(* Logix 5000 project; controller NSH_PLC2 vendor 1 type 14 code 167 rev 32.14; software revision 32.03 *)
// North State Hulling, PLC #2. Passes MCC#2 & #3 Motor Status & control to PLC #1

TASK MainTask (continuous, watchdog 500 ms) : MainProgram

MODULES
   Local : vendor 1 type 14 code 167 (ICP 1, Ethernet 192.168.2.253, rev 32.14)
      NSH_PLC1 : vendor 1 type 14 code 167 (ICP 0, rev 32.1)
      AOP_MCC3_3K : PowerFlex 525-EENET (Ethernet 192.168.3.10, rev 5.2, Output RPI 250 ms)
          : vendor 1 type 150 code 33279 (DSI 1, rev 3.1)
      AOP_MCC3_8K : PowerFlex 525-EENET (Ethernet 192.168.3.33, rev 5.2, Output RPI 250 ms)
          : vendor 1 type 150 code 33279 (DSI 1, rev 3.1)
      AOP_MCC2_21K : PowerFlex 525-EENET (Ethernet 192.168.2.116, rev 5.2, Output RPI 100 ms)
          : vendor 1 type 150 code 33279 (DSI 1, rev 3.1)
      AOP_MCC3_5K : PowerFlex 525-EENET (Ethernet 192.168.3.18, rev 5.2, Output RPI 250 ms)
          : vendor 1 type 150 code 33279 (DSI 1, rev 3.1)
      AOP_MCC3_2A : PowerFlex 525-EENET (Ethernet 192.168.3.3, rev 5.2, Output RPI 250 ms)
          : vendor 1 type 150 code 33279 (DSI 1, rev 3.1)
      AOP_MCC3_2K : PowerFlex 525-EENET (Ethernet 192.168.3.6, rev 5.2, Output RPI 250 ms)
          : vendor 1 type 150 code 33279 (DSI 1, rev 3.1)
      AOP_MCC3_3G : PowerFlex 525-EENET (Ethernet 192.168.3.9, rev 5.2, Output RPI 250 ms)
          : vendor 1 type 150 code 33279 (DSI 1, rev 3.1)
      AOP_MCC4_1E : PowerFlex 525-EENET (Ethernet 192.168.3.150, rev 6.1, Output RPI 100 ms)
          : vendor 1 type 150 code 33279 (DSI 1, rev 3.1)
      AOP_MCC3_4A : PowerFlex 525-EENET (Ethernet 192.168.3.11, rev 5.2, Output RPI 250 ms)
          : vendor 1 type 150 code 33279 (DSI 1, rev 3.1)
      AOP_MCC3_2D : PowerFlex 525-EENET (Ethernet 192.168.3.4, rev 5.2, Output RPI 250 ms)
          : vendor 1 type 150 code 33279 (DSI 1, rev 3.1)
      AOP_MCC2_9H : PowerFlex 525-EENET (Ethernet 192.168.2.43, rev 5.2, Output RPI 100 ms)
          : vendor 1 type 150 code 33279 (DSI 1, rev 3.1)
      AOP_MCC2_2K : PowerFlex 525-EENET (Ethernet 192.168.2.6, rev 5.2, Output RPI 250 ms)
          : vendor 1 type 150 code 33279 (DSI 1, rev 3.1)
      AOP_MCC3_4D : PowerFlex 525-EENET (Ethernet 192.168.3.12, rev 5.2, Output RPI 250 ms)
          : vendor 1 type 150 code 33279 (DSI 1, rev 3.1)
      AOP_MCC3_7G : PowerFlex 525-EENET (Ethernet 192.168.3.28, rev 5.2, Output RPI 250 ms)
          : vendor 1 type 150 code 33279 (DSI 1, rev 3.1)
      AOP_MCC3_3D : PowerFlex 525-EENET (Ethernet 192.168.3.8, rev 5.2, Output RPI 250 ms)
          : vendor 1 type 150 code 33279 (DSI 1, rev 3.1)
      AOP_MCC3_6D : PowerFlex 525-EENET (Ethernet 192.168.3.20, rev 5.2, Output RPI 250 ms)
          : vendor 1 type 150 code 33279 (DSI 1, rev 3.1)
      AOP_MCC4_2K : PowerFlex 525-EENET (Ethernet 192.168.3.155, rev 6.1, Output RPI 100 ms)
          : vendor 1 type 150 code 33279 (DSI 1, rev 3.1)
      AOP_MCC3_5G : PowerFlex 525-EENET (Ethernet 192.168.3.17, rev 5.2, Output RPI 250 ms)
          : vendor 1 type 150 code 33279 (DSI 1, rev 3.1)
      AOP_MCC3_6A : PowerFlex 525-EENET (Ethernet 192.168.3.19, rev 5.2, Output RPI 250 ms)
          : vendor 1 type 150 code 33279 (DSI 1, rev 3.1)
      AOP_MCC3_5D : PowerFlex 525-EENET (Ethernet 192.168.3.16, rev 5.2, Output RPI 250 ms)
      AOP_MCC2_2G : PowerFlex 525-EENET (Ethernet 192.168.2.5, rev 5.2, Output RPI 250 ms)
          : vendor 1 type 150 code 33279 (DSI 1, rev 3.1)
      AOP_MCC3_5A : PowerFlex 525-EENET (Ethernet 192.168.3.15, rev 5.2, Output RPI 250 ms)
          : vendor 1 type 150 code 33279 (DSI 1, rev 3.1)
      AOP_MCC3_7K : PowerFlex 525-EENET (Ethernet 192.168.3.29, rev 5.2, Output RPI 250 ms)
          : vendor 1 type 150 code 33279 (DSI 1, rev 3.1)
      AOP_MCC2_21G : PowerFlex 525-EENET (Ethernet 192.168.2.115, rev 5.2, Output RPI 250 ms)
          : vendor 1 type 150 code 33279 (DSI 1, rev 3.1)
      AOP_MCC3_2G : PowerFlex 525-EENET (Ethernet 192.168.3.5, rev 5.2, Output RPI 250 ms)
          : vendor 1 type 150 code 33279 (DSI 1, rev 3.1)
      AOP_MCC3_4G : PowerFlex 525-EENET (Ethernet 192.168.3.13, rev 5.2, Output RPI 250 ms)
          : vendor 1 type 150 code 33279 (DSI 1, rev 3.1)
      AOP_MCC2_2A : PowerFlex 525-EENET (Ethernet 192.168.2.3, rev 5.2, Output RPI 250 ms)
          : vendor 1 type 150 code 33279 (DSI 1, rev 3.1)
      AOP_MCC2_2D : PowerFlex 525-EENET (Ethernet 192.168.2.4, rev 5.2, Output RPI 250 ms)
          : vendor 1 type 150 code 33279 (DSI 1, rev 3.1)
      AOP_MCC3_8D : PowerFlex 525-EENET (Ethernet 192.168.3.31, rev 5.2, Output RPI 250 ms)
          : vendor 1 type 150 code 33279 (DSI 1, rev 3.1)
      AOP_MCC3_3A : PowerFlex 525-EENET (Ethernet 192.168.3.7, rev 5.2, Output RPI 250 ms)
          : vendor 1 type 150 code 33279 (DSI 1, rev 3.1)
      AOP_MCC4_2G : PowerFlex 525-EENET (Ethernet 192.168.3.154, rev 5.2, Output RPI 100 ms)
          : vendor 1 type 150 code 33279 (DSI 1, rev 3.1)
      AOP_MCC3_4K : PowerFlex 525-EENET (Ethernet 192.168.3.14, rev 5.2, Output RPI 250 ms)
          : vendor 1 type 150 code 33279 (DSI 1, rev 3.1)
      AOP_MCC2_13L_1 : vendor 1 type 12 code 237 (Ethernet 192.168.2.204, rev 10.1, Output RPI 1000 ms)
      AOP_MCC4_1L_1 : vendor 1 type 12 code 237 (Ethernet 192.168.3.210, rev 10.1, Output RPI 1000 ms)
      AOP_MCC2_9L_2 : vendor 1 type 12 code 243 (Ethernet 192.168.2.203, rev 10.1, Output RPI 1000 ms)
      AOP_MCC3_10L_2 : vendor 1 type 12 code 243 (Ethernet 192.168.3.203, rev 10.1, Output RPI 1000 ms)
      AOP_MCC3_15L_1 : vendor 1 type 12 code 237 (Ethernet 192.168.3.204, rev 10.1, Output RPI 1000 ms)
      AOP_MCC2_13L_2 : vendor 1 type 12 code 243 (Ethernet 192.168.2.205, rev 10.1, Output RPI 1000 ms)
      AOP_MCC3_15L_2 : vendor 1 type 12 code 243 (Ethernet 192.168.3.205, rev 10.1, Output RPI 1000 ms)
      AOP_MCC4_1L_2 : vendor 1 type 12 code 243 (Ethernet 192.168.3.211, rev 10.1, Output RPI 1000 ms)
      AOP_MCC2_5L_1 : vendor 1 type 12 code 237 (Ethernet 192.168.2.200, rev 10.1, Output RPI 1000 ms)
      AOP_MCC3_6L_2 : vendor 1 type 12 code 243 (Ethernet 192.168.3.201, rev 10.1, Output RPI 1000 ms)
      AOP_MCC3_20L_1 : vendor 1 type 12 code 237 (Ethernet 192.168.3.208, rev 10.1, Output RPI 1000 ms)
      AOP_MCC2_9L_1 : vendor 1 type 12 code 237 (Ethernet 192.168.2.202, rev 10.1, Output RPI 1000 ms)
      AOP_MCC2_20L_2 : vendor 1 type 12 code 243 (Ethernet 192.168.2.209, rev 10.1, Output RPI 1000 ms)
      AOP_MCC3_19L_2 : vendor 1 type 12 code 243 (Ethernet 192.168.3.207, rev 10.1, Output RPI 1000 ms)
      AOP_MCC3_20L_2 : vendor 1 type 12 code 243 (Ethernet 192.168.3.209, rev 10.1, Output RPI 1000 ms)
      AOP_MCC2_5L_2 : vendor 1 type 12 code 243 (Ethernet 192.168.2.201, rev 10.1, Output RPI 1000 ms)
      AOP_MCC2_20L_1 : vendor 1 type 12 code 237 (Ethernet 192.168.2.208, rev 10.1, Output RPI 1000 ms)
      AOP_MCC3_6L_1 : vendor 1 type 12 code 237 (Ethernet 192.168.3.200, rev 10.1, Output RPI 1000 ms)
      AOP_MCC2_17L_2 : vendor 1 type 12 code 243 (Ethernet 192.168.2.207, rev 10.1, Output RPI 1000 ms)
      AOP_MCC2_17L_1 : vendor 1 type 12 code 237 (Ethernet 192.168.2.206, rev 10.1, Output RPI 1000 ms)
      AOP_MCC3_19L_1 : vendor 1 type 12 code 237 (Ethernet 192.168.3.206, rev 10.1, Output RPI 1000 ms)
      AOP_MCC3_10L_1 : vendor 1 type 12 code 237 (Ethernet 192.168.3.202, rev 10.1, Output RPI 1000 ms)
      AOP_MCC3_16G : 193-ECM-ETR (Ethernet 192.168.3.78, rev 7.17, StandardDataDriven RPI 100 ms)
      AOP_MCC2_4C : 193-ECM-ETR (Ethernet 192.168.2.14, rev 7.17, StandardDataDriven RPI 100 ms)
      AOP_MCC2_21E : 193-ECM-ETR (Ethernet 192.168.2.114, rev 7.17, StandardDataDriven RPI 100 ms)
      AOP_MCC3_13C : 193-ECM-ETR (Ethernet 192.168.3.57, rev 7.17, StandardDataDriven RPI 100 ms)
      AOP_MCC3_18C : 193-ECM-ETR (Ethernet 192.168.3.88, rev 7.17, StandardDataDriven RPI 100 ms)
      AOP_MCC3_13A : 193-ECM-ETR (Ethernet 192.168.3.56, rev 7.17, StandardDataDriven RPI 100 ms)
      AOP_MCC3_15C : 193-ECM-ETR (Ethernet 192.168.3.69, rev 7.17, StandardDataDriven RPI 100 ms)
      AOP_MCC3_6G : 193-ECM-ETR (Ethernet 192.168.3.21, rev 7.17, StandardDataDriven RPI 100 ms)
      AOP_MCC2_4L : 193-ECM-ETR (Ethernet 192.168.2.18, rev 7.17, StandardDataDriven RPI 100 ms)
      AOP_MCC3_11A : 193-ECM-ETR (Ethernet 192.168.3.44, rev 7.17, StandardDataDriven RPI 100 ms)
      AOP_MCC2_10A : 193-ECM-ETR (Ethernet 192.168.2.46, rev 7.17, StandardDataDriven RPI 100 ms)
      AOP_MCC2_13J : 193-ECM-ETR (Ethernet 192.168.2.68, rev 7.17, StandardDataDriven RPI 100 ms)
      AOP_MCC4_4A : 193-ECM-ETR (Ethernet 192.168.3.162, rev 7.17, StandardDataDriven RPI 100 ms)
      AOP_MCC2_4G : 193-ECM-ETR (Ethernet 192.168.2.16, rev 7.17, StandardDataDriven RPI 100 ms)
      AOP_MCC2_8D : 193-ECM-ETR (Ethernet 192.168.2.37, rev 7.17, StandardDataDriven RPI 100 ms)
      AOP_MCC4_5C : 193-ECM-ETR (Ethernet 192.168.3.169, rev 7.17, StandardDataDriven RPI 100 ms)
      AOP_MCC3_16E : 193-ECM-ETR (Ethernet 192.168.3.77, rev 7.17, StandardDataDriven RPI 100 ms)
      AOP_MCC3_10J : 193-ECM-ETR (Ethernet 192.168.3.43, rev 7.17, StandardDataDriven RPI 100 ms)
      AOP_MCC2_3A : 193-ECM-ETR (Ethernet 192.168.2.7, rev 7.17, StandardDataDriven RPI 100 ms)
      AOP_MCC3_13G : 193-ECM-ETR (Ethernet 192.168.3.59, rev 7.17, StandardDataDriven RPI 100 ms)
      AOP_MCC2_3C : 193-ECM-ETR (Ethernet 192.168.2.8, rev 7.17, StandardDataDriven RPI 100 ms)
      AOP_MCC3_12G : 193-ECM-ETR (Ethernet 192.168.3.53, rev 7.17, StandardDataDriven RPI 100 ms)
      AOP_MCC4_4L : 193-ECM-ETR (Ethernet 192.168.3.167, rev 7.17, StandardDataDriven RPI 100 ms)
      AOP_MCC2_14E : 193-ECM-ETR (Ethernet 192.168.2.73, rev 7.17, StandardDataDriven RPI 100 ms)
      AOP_MCC3_21C : 193-ECM-ETR (Ethernet 192.168.3.106, rev 7.17, StandardDataDriven RPI 100 ms)
      AOP_MCC3_21E : 193-ECM-ETR (Ethernet 192.168.3.107, rev 7.17, StandardDataDriven RPI 100 ms)
      AOP_MCC3_20G : 193-ECM-ETR (Ethernet 192.168.3.103, rev 7.17, StandardDataDriven RPI 100 ms)
      AOP_MCC2_12J : 193-ECM-ETR (Ethernet 192.168.2.62, rev 7.17, StandardDataDriven RPI 100 ms)
      AOP_MCC3_12J : 193-ECM-ETR (Ethernet 192.168.3.54, rev 7.17, StandardDataDriven RPI 100 ms)
      AOP_MCC3_15E : 193-ECM-ETR (Ethernet 192.168.3.70, rev 7.17, StandardDataDriven RPI 100 ms)
      AOP_MCC3_19C : 193-ECM-ETR (Ethernet 192.168.3.94, rev 7.17, StandardDataDriven RPI 100 ms)
      AOP_MCC4_4G : 193-ECM-ETR (Ethernet 192.168.3.165, rev 7.17, StandardDataDriven RPI 100 ms)
      AOP_MCC3_8H : 193-ECM-ETR (Ethernet 192.168.3.32, rev 7.17, StandardDataDriven RPI 100 ms)
      AOP_MCC2_11G : 193-ECM-ETR (Ethernet 192.168.2.55, rev 7.17, StandardDataDriven RPI 100 ms)
      AOP_MCC2_17C : 193-ECM-ETR (Ethernet 192.168.2.90, rev 7.17, StandardDataDriven RPI 100 ms)
      AOP_MCC3_14G : 193-ECM-ETR (Ethernet 192.168.3.65, rev 7.17, StandardDataDriven RPI 100 ms)
      AOP_MCC4_2A : 193-ECM-ETR (Ethernet 192.168.3.151, rev 7.17, StandardDataDriven RPI 100 ms)
      AOP_MCC3_22E : 193-ECM-ETR (Ethernet 192.168.3.112, rev 7.17, StandardDataDriven RPI 100 ms)
      AOP_MCC3_15G : 193-ECM-ETR (Ethernet 192.168.3.71, rev 7.17, StandardDataDriven RPI 100 ms)
      AOP_MCC2_13C : 193-ECM-ETR (Ethernet 192.168.2.65, rev 7.17, StandardDataDriven RPI 100 ms)
      AOP_MCC2_3J : 193-ECM-ETR (Ethernet 192.168.2.11, rev 7.17, StandardDataDriven RPI 100 ms)
      AOP_MCC3_17G : 193-ECM-ETR (Ethernet 192.168.3.84, rev 7.17, StandardDataDriven RPI 250 ms)
      AOP_MCC3_17A : 193-ECM-ETR (Ethernet 192.168.3.81, rev 7.17, StandardDataDriven RPI 100 ms)
      AOP_MCC3_19A : 193-ECM-ETR (Ethernet 192.168.3.93, rev 7.17, StandardDataDriven RPI 100 ms)
      AOP_MCC2_16E : 193-ECM-ETR (Ethernet 192.168.2.85, rev 7.17, StandardDataDriven RPI 100 ms)
      AOP_MCC2_10C : 193-ECM-ETR (Ethernet 192.168.2.47, rev 7.17, StandardDataDriven RPI 100 ms)
      AOP_MCC3_21G : 193-ECM-ETR (Ethernet 192.168.3.108, rev 7.17, StandardDataDriven RPI 100 ms)
      AOP_MCC2_8H : 193-ECM-ETR (Ethernet 192.168.2.39, rev 7.17, StandardDataDriven RPI 100 ms)
      AOP_MCC2_6C : 193-ECM-ETR (Ethernet 192.168.2.27, rev 7.17, StandardDataDriven RPI 100 ms)
      AOP_MCC4_3G : 193-ECM-ETR (Ethernet 192.168.3.159, rev 7.17, StandardDataDriven RPI 100 ms)
      AOP_MCC2_16C : 193-ECM-ETR (Ethernet 192.168.2.84, rev 7.17, StandardDataDriven RPI 100 ms)
      AOP_MCC3_18G : 193-ECM-ETR (Ethernet 192.168.3.90, rev 7.17, StandardDataDriven RPI 100 ms)
      AOP_MCC2_8F : 193-ECM-ETR (Ethernet 192.168.2.38, rev 7.17, StandardDataDriven RPI 100 ms)
      AOP_MCC2_13E : 193-ECM-ETR (Ethernet 192.168.2.66, rev 7.17, StandardDataDriven RPI 100 ms)
      AOP_MCC3_12L : 193-ECM-ETR (Ethernet 192.168.3.55, rev 7.17, StandardDataDriven RPI 100 ms)
      AOP_MCC2_18J : 193-ECM-ETR (Ethernet 192.168.2.100, rev 7.17, StandardDataDriven RPI 100 ms)
      AOP_MCC2_20J : 193-ECM-ETR (Ethernet 192.168.2.111, rev 7.17, StandardDataDriven RPI 100 ms)
      AOP_MCC2_15G : 193-ECM-ETR (Ethernet 192.168.2.80, rev 7.17, StandardDataDriven RPI 100 ms)
      AOP_MCC3_19G : 193-ECM-ETR (Ethernet 192.168.3.96, rev 7.17, StandardDataDriven RPI 100 ms)
      AOP_MCC4_2E : 193-ECM-ETR (Ethernet 192.168.3.153, rev 7.17, StandardDataDriven RPI 100 ms)
      AOP_MCC2_19C : 193-ECM-ETR (Ethernet 192.168.2.103, rev 7.17, StandardDataDriven RPI 100 ms)
      AOP_MCC2_15J : 193-ECM-ETR (Ethernet 192.168.2.81, rev 7.17, StandardDataDriven RPI 100 ms)
      AOP_MCC3_12A : 193-ECM-ETR (Ethernet 192.168.3.50, rev 7.17, StandardDataDriven RPI 100 ms)
      AOP_MCC3_11G : 193-ECM-ETR (Ethernet 192.168.3.46, rev 7.17, StandardDataDriven RPI 100 ms)
      AOP_MCC3_13L : 193-ECM-ETR (Ethernet 192.168.3.61, rev 7.17, StandardDataDriven RPI 100 ms)
      AOP_MCC2_11J : 193-ECM-ETR (Ethernet 192.168.2.56, rev 7.17, StandardDataDriven RPI 100 ms)
      AOP_MCC3_6J : 193-ECM-ETR (Ethernet 192.168.3.22, rev 7.17, StandardDataDriven RPI 100 ms)
      AOP_MCC3_10G : 193-ECM-ETR (Ethernet 192.168.3.42, rev 7.17, StandardDataDriven RPI 100 ms)
      AOP_MCC2_16L : 193-ECM-ETR (Ethernet 192.168.2.88, rev 7.17, StandardDataDriven RPI 100 ms)
      AOP_MCC2_18C : 193-ECM-ETR (Ethernet 192.168.2.97, rev 7.17, StandardDataDriven RPI 100 ms)
      AOP_MCC2_14G : 193-ECM-ETR (Ethernet 192.168.2.74, rev 7.17, StandardDataDriven RPI 100 ms)
      AOP_MCC2_7G : 193-ECM-ETR (Ethernet 192.168.2.34, rev 7.17, StandardDataDriven RPI 100 ms)
      AOP_MCC2_19E : 193-ECM-ETR (Ethernet 192.168.2.104, rev 7.17, StandardDataDriven RPI 100 ms)
      AOP_MCC2_15E : 193-ECM-ETR (Ethernet 192.168.2.79, rev 7.17, StandardDataDriven RPI 100 ms)
      AOP_MCC3_21A : 193-ECM-ETR (Ethernet 192.168.3.105, rev 7.17, StandardDataDriven RPI 100 ms)
      AOP_MCC2_5G : 193-ECM-ETR (Ethernet 192.168.2.22, rev 7.17, StandardDataDriven RPI 100 ms)
      AOP_MCC3_18L : 193-ECM-ETR (Ethernet 192.168.3.92, rev 7.17, StandardDataDriven RPI 100 ms)
      AOP_MCC2_10E : 193-ECM-ETR (Ethernet 192.168.2.48, rev 7.17, StandardDataDriven RPI 100 ms)
      AOP_MCC2_3G : 193-ECM-ETR (Ethernet 192.168.2.10, rev 7.17, StandardDataDriven RPI 100 ms)
      AOP_MCC3_16J : 193-ECM-ETR (Ethernet 192.168.3.79, rev 7.17, StandardDataDriven RPI 100 ms)
      AOP_MCC3_7E : 193-ECM-ETR (Ethernet 192.168.3.27, rev 7.17, StandardDataDriven RPI 100 ms)
      AOP_MCC2_13A : 193-ECM-ETR (Ethernet 192.168.2.64, rev 7.17, StandardDataDriven RPI 100 ms)
      AOP_MCC3_19J : 193-ECM-ETR (Ethernet 192.168.3.97, rev 7.17, StandardDataDriven RPI 100 ms)
      AOP_MCC3_21J : 193-ECM-ETR (Ethernet 192.168.3.109, rev 7.17, StandardDataDriven RPI 100 ms)
      AOP_MCC2_13G : 193-ECM-ETR (Ethernet 192.168.2.67, rev 7.17, StandardDataDriven RPI 100 ms)
      AOP_MCC2_7K : 193-ECM-ETR (Ethernet 192.168.2.35, rev 7.17, StandardDataDriven RPI 100 ms)
      AOP_MCC3_20C : 193-ECM-ETR (Ethernet 192.168.3.101, rev 7.17, StandardDataDriven RPI 100 ms)
      AOP_MCC2_18L : 193-ECM-ETR (Ethernet 192.168.2.101, rev 7.17, StandardDataDriven RPI 100 ms)
      AOP_MCC2_3E : 193-ECM-ETR (Ethernet 192.168.2.9, rev 7.17, StandardDataDriven RPI 100 ms)
      AOP_MCC2_6L : 193-ECM-ETR (Ethernet 192.168.2.31, rev 7.17, StandardDataDriven RPI 100 ms)
      AOP_MCC2_16A : 193-ECM-ETR (Ethernet 192.168.2.83, rev 7.17, StandardDataDriven RPI 100 ms)
      AOP_MCC3_9L : 193-ECM-ETR (Ethernet 192.168.3.39, rev 7.17, StandardDataDriven RPI 100 ms)
      AOP_MCC2_12A : 193-ECM-ETR (Ethernet 192.168.2.58, rev 7.17, StandardDataDriven RPI 100 ms)
      AOP_MCC3_18J : 193-ECM-ETR (Ethernet 192.168.3.91, rev 7.17, StandardDataDriven RPI 100 ms)
      AOP_MCC4_4J : 193-ECM-ETR (Ethernet 192.168.3.166, rev 7.17, StandardDataDriven RPI 100 ms)
      AOP_MCC3_14L : 193-ECM-ETR (Ethernet 192.168.3.67, rev 7.17, StandardDataDriven RPI 100 ms)
      AOP_MCC3_12C : 193-ECM-ETR (Ethernet 192.168.3.51, rev 7.17, StandardDataDriven RPI 100 ms)
      AOP_MCC2_3L : 193-ECM-ETR (Ethernet 192.168.2.12, rev 7.17, StandardDataDriven RPI 100 ms)
      AOP_MCC3_9G : 193-ECM-ETR (Ethernet 192.168.3.37, rev 7.17, StandardDataDriven RPI 100 ms)
      AOP_MCC3_17C : 193-ECM-ETR (Ethernet 192.168.3.82, rev 7.17, StandardDataDriven RPI 100 ms)
      AOP_MCC3_17L : 193-ECM-ETR (Ethernet 192.168.3.86, rev 7.17, StandardDataDriven RPI 100 ms)
      AOP_MCC4_4C : 193-ECM-ETR (Ethernet 192.168.3.163, rev 7.17, StandardDataDriven RPI 100 ms)
      AOP_MCC2_4E : 193-ECM-ETR (Ethernet 192.168.2.15, rev 7.17, StandardDataDriven RPI 100 ms)
      AOP_MCC3_9C : 193-ECM-ETR (Ethernet 192.168.3.35, rev 7.17, StandardDataDriven RPI 100 ms)
      AOP_MCC2_17A : 193-ECM-ETR (Ethernet 192.168.2.89, rev 7.17, StandardDataDriven RPI 100 ms)
      AOP_MCC3_9E : 193-ECM-ETR (Ethernet 192.168.3.36, rev 7.17, StandardDataDriven RPI 100 ms)
      AOP_MCC3_18E : 193-ECM-ETR (Ethernet 192.168.3.89, rev 7.17, StandardDataDriven RPI 100 ms)
      AOP_MCC2_11C : 193-ECM-ETR (Ethernet 192.168.2.53, rev 7.17, StandardDataDriven RPI 100 ms)
      AOP_MCC2_18E : 193-ECM-ETR (Ethernet 192.168.2.98, rev 7.17, StandardDataDriven RPI 100 ms)
      AOP_MCC2_5A : 193-ECM-ETR (Ethernet 192.168.2.19, rev 7.17, StandardDataDriven RPI 100 ms)
      AOP_MCC3_16L : 193-ECM-ETR (Ethernet 192.168.3.80, rev 7.17, StandardDataDriven RPI 100 ms)
      AOP_MCC2_19J : 193-ECM-ETR (Ethernet 192.168.2.106, rev 7.17, StandardDataDriven RPI 100 ms)
      AOP_MCC2_10G : 193-ECM-ETR (Ethernet 192.168.2.49, rev 7.17, StandardDataDriven RPI 100 ms)
      AOP_MCC4_3C : 193-ECM-ETR (Ethernet 192.168.3.157, rev 7.17, StandardDataDriven RPI 100 ms)
      AOP_MCC4_2C : 193-ECM-ETR (Ethernet 192.168.3.152, rev 7.17, StandardDataDriven RPI 100 ms)
      AOP_MCC2_19A : 193-ECM-ETR (Ethernet 192.168.2.102, rev 7.17, StandardDataDriven RPI 100 ms)
      AOP_MCC2_20G : 193-ECM-ETR (Ethernet 192.168.2.110, rev 7.17, StandardDataDriven RPI 100 ms)
      AOP_MCC3_14J : 193-ECM-ETR (Ethernet 192.168.3.66, rev 7.17, StandardDataDriven RPI 100 ms)
      AOP_MCC2_10L : 193-ECM-ETR (Ethernet 192.168.2.51, rev 7.17, StandardDataDriven RPI 100 ms)
      AOP_MCC3_15A : 193-ECM-ETR (Ethernet 192.168.3.68, rev 7.17, StandardDataDriven RPI 100 ms)
      AOP_MCC2_14L : 193-ECM-ETR (Ethernet 192.168.2.76, rev 7.17, StandardDataDriven RPI 100 ms)
      AOP_MCC4_3E : 193-ECM-ETR (Ethernet 192.168.3.158, rev 7.17, StandardDataDriven RPI 100 ms)
      AOP_MCC2_19L : 193-ECM-ETR (Ethernet 192.168.2.107, rev 7.17, StandardDataDriven RPI 100 ms)
      AOP_MCC2_17J : 193-ECM-ETR (Ethernet 192.168.2.93, rev 7.17, StandardDataDriven RPI 100 ms)
      AOP_MCC3_14A : 193-ECM-ETR (Ethernet 192.168.3.62, rev 7.17, StandardDataDriven RPI 100 ms)
      AOP_MCC3_14E : 193-ECM-ETR (Ethernet 192.168.3.64, rev 7.17, StandardDataDriven RPI 100 ms)
      AOP_MCC2_4A : 193-ECM-ETR (Ethernet 192.168.2.13, rev 7.17, StandardDataDriven RPI 100 ms)
      AOP_MCC4_4E : 193-ECM-ETR (Ethernet 192.168.3.164, rev 7.17, StandardDataDriven RPI 100 ms)
      AOP_MCC2_10J : 193-ECM-ETR (Ethernet 192.168.2.50, rev 7.17, StandardDataDriven RPI 100 ms)
      AOP_MCC3_20A : 193-ECM-ETR (Ethernet 192.168.3.100, rev 7.17, StandardDataDriven RPI 100 ms)
      AOP_MCC2_6G : 193-ECM-ETR (Ethernet 192.168.2.29, rev 7.17, StandardDataDriven RPI 100 ms)
      AOP_MCC3_16A : 193-ECM-ETR (Ethernet 192.168.3.75, rev 7.17, StandardDataDriven RPI 100 ms)
      AOP_MCC2_14J : 193-ECM-ETR (Ethernet 192.168.2.75, rev 7.17, StandardDataDriven RPI 100 ms)
      AOP_MCC2_6A : 193-ECM-ETR (Ethernet 192.168.2.26, rev 7.17, StandardDataDriven RPI 100 ms)
      AOP_MCC2_17G : 193-ECM-ETR (Ethernet 192.168.2.92, rev 7.17, StandardDataDriven RPI 100 ms)
      AOP_MCC2_17E : 193-ECM-ETR (Ethernet 192.168.2.91, rev 7.17, StandardDataDriven RPI 100 ms)
      AOP_MCC2_20C : 193-ECM-ETR (Ethernet 192.168.2.108, rev 7.17, StandardDataDriven RPI 100 ms)
      AOP_MCC3_18A : 193-ECM-ETR (Ethernet 192.168.3.87, rev 7.17, StandardDataDriven RPI 100 ms)
      AOP_MCC2_6J : 193-ECM-ETR (Ethernet 192.168.2.30, rev 7.17, StandardDataDriven RPI 100 ms)
      AOP_MCC3_17J : 193-ECM-ETR (Ethernet 192.168.3.85, rev 7.17, StandardDataDriven RPI 100 ms)
      AOP_MCC2_12L : 193-ECM-ETR (Ethernet 192.168.2.63, rev 7.17, StandardDataDriven RPI 100 ms)
      AOP_MCC2_15L : 193-ECM-ETR (Ethernet 192.168.2.82, rev 7.17, StandardDataDriven RPI 100 ms)
      AOP_MCC3_19E : 193-ECM-ETR (Ethernet 192.168.3.95, rev 7.17, StandardDataDriven RPI 100 ms)
      AOP_MCC2_8K : 193-ECM-ETR (Ethernet 192.168.2.40, rev 7.17, StandardDataDriven RPI 250 ms)
      AOP_MCC3_21L : 193-ECM-ETR (Ethernet 192.168.3.110, rev 7.17, StandardDataDriven RPI 100 ms)
      AOP_MCC2_11A : 193-ECM-ETR (Ethernet 192.168.2.52, rev 7.17, StandardDataDriven RPI 100 ms)
      AOP_MCC2_14C : 193-ECM-ETR (Ethernet 192.168.2.72, rev 7.17, StandardDataDriven RPI 100 ms)
      AOP_MCC2_14A : 193-ECM-ETR (Ethernet 192.168.2.71, rev 7.17, StandardDataDriven RPI 100 ms)
      AOP_MCC2_4J : 193-ECM-ETR (Ethernet 192.168.2.17, rev 7.17, StandardDataDriven RPI 100 ms)
      AOP_MCC2_11E : 193-ECM-ETR (Ethernet 192.168.2.54, rev 7.17, StandardDataDriven RPI 100 ms)
      AOP_MCC2_6E : 193-ECM-ETR (Ethernet 192.168.2.28, rev 7.17, StandardDataDriven RPI 100 ms)
      AOP_MCC2_21C : 193-ECM-ETR (Ethernet 192.168.2.113, rev 7.17, StandardDataDriven RPI 100 ms)
      AOP_MCC3_13J : 193-ECM-ETR (Ethernet 192.168.3.60, rev 7.17, StandardDataDriven RPI 100 ms)
      AOP_MCC3_7C : 193-ECM-ETR (Ethernet 192.168.3.26, rev 7.17, StandardDataDriven RPI 100 ms)
      AOP_MCC3_10A : 193-ECM-ETR (Ethernet 192.168.3.40, rev 7.17, StandardDataDriven RPI 100 ms)
      AOP_MCC2_9F : 193-ECM-ETR (Ethernet 192.168.2.42, rev 7.17, StandardDataDriven RPI 100 ms)
      AOP_MCC2_8B : 193-ECM-ETR (Ethernet 192.168.2.36, rev 7.17, StandardDataDriven RPI 100 ms)
      AOP_MCC3_20E : 193-ECM-ETR (Ethernet 192.168.3.102, rev 7.17, StandardDataDriven RPI 100 ms)
      AOP_MCC3_13E : 193-ECM-ETR (Ethernet 192.168.3.58, rev 7.17, StandardDataDriven RPI 100 ms)
      AOP_MCC3_16C : 193-ECM-ETR (Ethernet 192.168.3.76, rev 7.17, StandardDataDriven RPI 100 ms)
      AOP_MCC2_5E : 193-ECM-ETR (Ethernet 192.168.2.21, rev 7.17, StandardDataDriven RPI 100 ms)
      AOP_MCC3_9A : 193-ECM-ETR (Ethernet 192.168.3.34, rev 7.17, StandardDataDriven RPI 100 ms)
      AOP_MCC2_15A : 193-ECM-ETR (Ethernet 192.168.2.77, rev 7.17, StandardDataDriven RPI 100 ms)
      AOP_MCC2_5C : 193-ECM-ETR (Ethernet 192.168.2.20, rev 7.17, StandardDataDriven RPI 100 ms)
      AOP_MCC2_12G : 193-ECM-ETR (Ethernet 192.168.2.61, rev 7.17, StandardDataDriven RPI 100 ms)
      AOP_MCC3_22C : 193-ECM-ETR (Ethernet 192.168.3.111, rev 7.17, StandardDataDriven RPI 100 ms)
      AOP_MCC2_11L : 193-ECM-ETR (Ethernet 192.168.2.57, rev 7.17, StandardDataDriven RPI 100 ms)
      AOP_MCC2_16J : 193-ECM-ETR (Ethernet 192.168.2.87, rev 7.17, StandardDataDriven RPI 100 ms)
      AOP_MCC2_12C : 193-ECM-ETR (Ethernet 192.168.2.59, rev 7.17, StandardDataDriven RPI 100 ms)
      AOP_MCC4_3A : 193-ECM-ETR (Ethernet 192.168.3.156, rev 7.17, StandardDataDriven RPI 100 ms)
      AOP_MCC2_7D : 193-ECM-ETR (Ethernet 192.168.2.33, rev 7.17, StandardDataDriven RPI 100 ms)
      AOP_MCC3_8A : 193-ECM-ETR (Ethernet 192.168.3.30, rev 7.17, StandardDataDriven RPI 100 ms)
      AOP_MCC2_7A : 193-ECM-ETR (Ethernet 192.168.2.32, rev 7.17, StandardDataDriven RPI 100 ms)
      AOP_MCC2_15C : 193-ECM-ETR (Ethernet 192.168.2.78, rev 7.17, StandardDataDriven RPI 150 ms)
      AOP_MCC2_12E : 193-ECM-ETR (Ethernet 192.168.2.60, rev 7.17, StandardDataDriven RPI 100 ms)
      AOP_MCC2_20E : 193-ECM-ETR (Ethernet 192.168.2.109, rev 7.17, StandardDataDriven RPI 100 ms)
      AOP_MCC4_3L : 193-ECM-ETR (Ethernet 192.168.3.161, rev 7.17, StandardDataDriven RPI 100 ms)
      AOP_MCC2_18A : 193-ECM-ETR (Ethernet 192.168.2.96, rev 7.17, StandardDataDriven RPI 100 ms)
      AOP_MCC3_20J : 193-ECM-ETR (Ethernet 192.168.3.104, rev 7.17, StandardDataDriven RPI 100 ms)
      AOP_MCC2_9D : 193-ECM-ETR (Ethernet 192.168.2.41, rev 7.17, StandardDataDriven RPI 100 ms)
      AOP_MCC2_19G : 193-ECM-ETR (Ethernet 192.168.2.105, rev 7.17, StandardDataDriven RPI 100 ms)
      AOP_MCC2_21A : 193-ECM-ETR (Ethernet 192.168.2.112, rev 7.17, StandardDataDriven RPI 100 ms)
      AOP_MCC4_5A : 193-ECM-ETR (Ethernet 192.168.3.168, rev 7.17, StandardDataDriven RPI 100 ms)
      AOP_MCC3_9J : 193-ECM-ETR (Ethernet 192.168.3.38, rev 7.17, StandardDataDriven RPI 100 ms)
      AOP_MCC3_11J : 193-ECM-ETR (Ethernet 192.168.3.47, rev 7.17, StandardDataDriven RPI 100 ms)
      AOP_MCC3_17E : 193-ECM-ETR (Ethernet 192.168.3.83, rev 7.17, StandardDataDriven RPI 100 ms)
      AOP_MCC4_3J : 193-ECM-ETR (Ethernet 192.168.3.160, rev 7.17, StandardDataDriven RPI 100 ms)
      AOP_MCC2_18G : 193-ECM-ETR (Ethernet 192.168.2.99, rev 7.17, StandardDataDriven RPI 100 ms)
      AOP_MCC3_14C : 193-ECM-ETR (Ethernet 192.168.3.63, rev 7.17, StandardDataDriven RPI 100 ms)
      AOP_MCC2_5J : 193-ECM-ETR (Ethernet 192.168.2.23, rev 7.17, StandardDataDriven RPI 100 ms)
      AOP_MCC2_16G : 193-ECM-ETR (Ethernet 192.168.2.86, rev 7.17, StandardDataDriven RPI 100 ms)
      AOP_MCC3_11D : 193-ECM-ETR (Ethernet 192.168.3.45, rev 7.17, StandardDataDriven RPI 100 ms)
      AOP_MCC3_10D : 193-ECM-ETR (Ethernet 192.168.3.41, rev 7.17, StandardDataDriven RPI 100 ms)
      AOP_MCC3_7A : 193-ECM-ETR (Ethernet 192.168.3.25, rev 7.17, StandardDataDriven RPI 100 ms)
      AOP_MCC3_15J : 193-ECM-ETR (Ethernet 192.168.3.72, rev 7.17, StandardDataDriven RPI 100 ms)
      AOP_MCC3_12E : 193-ECM-ETR (Ethernet 192.168.3.52, rev 7.17, StandardDataDriven RPI 100 ms)
END_MODULES

TYPE MotorControlUDT :   // Control Bits & Speed 0->100% to PLC2 for MCC2 & MCC3
STRUCT
   CommandBits : DINT;   // Bit 0=Run 1 = Fault Reset
   Speed : DINT;   // 0->100% Converted to VFD Reference in PLC2, MotorToPF525 AOI
   Spare : DINT;   // Spare DINT
END_STRUCT
END_TYPE

TYPE MotorsControlUDT :
STRUCT
   MCC2_2A : MotorControlUDT;
   MCC2_2D : MotorControlUDT;
   MCC2_2G : MotorControlUDT;
   MCC2_2K : MotorControlUDT;
   MCC2_3A : MotorControlUDT;
   MCC2_3C : MotorControlUDT;
   MCC2_3E : MotorControlUDT;
   MCC2_3G : MotorControlUDT;
   MCC2_3J : MotorControlUDT;
   MCC2_3L : MotorControlUDT;
   MCC2_4A : MotorControlUDT;
   MCC2_4C : MotorControlUDT;
   MCC2_4E : MotorControlUDT;
   MCC2_4G : MotorControlUDT;
   MCC2_4J : MotorControlUDT;
   MCC2_4L : MotorControlUDT;
   MCC2_5A : MotorControlUDT;
   MCC2_5C : MotorControlUDT;
   MCC2_5E : MotorControlUDT;
   MCC2_5G : MotorControlUDT;
   MCC2_5J : MotorControlUDT;
   MCC2_6A : MotorControlUDT;
   MCC2_6C : MotorControlUDT;
   MCC2_6E : MotorControlUDT;
   MCC2_6G : MotorControlUDT;
   MCC2_6J : MotorControlUDT;
   MCC2_6L : MotorControlUDT;
   MCC2_7A : MotorControlUDT;
   MCC2_7D : MotorControlUDT;
   MCC2_7G : MotorControlUDT;
   MCC2_7K : MotorControlUDT;
   MCC2_8B : MotorControlUDT;
   MCC2_8D : MotorControlUDT;
   MCC2_8F : MotorControlUDT;
   MCC2_8H : MotorControlUDT;
   MCC2_8K : MotorControlUDT;
   MCC2_9D : MotorControlUDT;
   MCC2_9F : MotorControlUDT;
   MCC2_9H : MotorControlUDT;
   MCC2_10A : MotorControlUDT;
   MCC2_10C : MotorControlUDT;
   MCC2_10E : MotorControlUDT;
   MCC2_10G : MotorControlUDT;
   MCC2_10J : MotorControlUDT;
   MCC2_10L : MotorControlUDT;
   MCC2_11A : MotorControlUDT;
   MCC2_11C : MotorControlUDT;
   MCC2_11E : MotorControlUDT;
   MCC2_11G : MotorControlUDT;
   MCC2_11J : MotorControlUDT;
   MCC2_11L : MotorControlUDT;
   MCC2_12A : MotorControlUDT;
   MCC2_12C : MotorControlUDT;
   MCC2_12E : MotorControlUDT;
   MCC2_12G : MotorControlUDT;
   MCC2_12J : MotorControlUDT;
   MCC2_12L : MotorControlUDT;
   MCC2_13A : MotorControlUDT;
   MCC2_13C : MotorControlUDT;
   MCC2_13E : MotorControlUDT;
   MCC2_13G : MotorControlUDT;
   MCC2_13J : MotorControlUDT;
   MCC2_14A : MotorControlUDT;
   MCC2_14C : MotorControlUDT;
   MCC2_14E : MotorControlUDT;
   MCC2_14G : MotorControlUDT;
   MCC2_14J : MotorControlUDT;
   MCC2_14L : MotorControlUDT;
   MCC2_15A : MotorControlUDT;
   MCC2_15C : MotorControlUDT;
   MCC2_15E : MotorControlUDT;
   MCC2_15G : MotorControlUDT;
   MCC2_15J : MotorControlUDT;
   MCC2_15L : MotorControlUDT;
   MCC2_16A : MotorControlUDT;
   MCC2_16C : MotorControlUDT;
   MCC2_16E : MotorControlUDT;
   MCC2_16G : MotorControlUDT;
   MCC2_16J : MotorControlUDT;
   MCC2_16L : MotorControlUDT;
   MCC2_17A : MotorControlUDT;
   MCC2_17C : MotorControlUDT;
   MCC2_17E : MotorControlUDT;
   MCC2_17G : MotorControlUDT;
   MCC2_17J : MotorControlUDT;
   MCC2_18A : MotorControlUDT;
   MCC2_18C : MotorControlUDT;
   MCC2_18E : MotorControlUDT;
   MCC2_18G : MotorControlUDT;
   MCC2_18J : MotorControlUDT;
   MCC2_18L : MotorControlUDT;
   MCC2_19A : MotorControlUDT;
   MCC2_19C : MotorControlUDT;
   MCC2_19E : MotorControlUDT;
   MCC2_19G : MotorControlUDT;
   MCC2_19J : MotorControlUDT;
   MCC2_19L : MotorControlUDT;
   MCC2_20C : MotorControlUDT;
   MCC2_20E : MotorControlUDT;
   MCC2_20G : MotorControlUDT;
   MCC2_20J : MotorControlUDT;
   MCC2_21A : MotorControlUDT;
   MCC2_21C : MotorControlUDT;
   MCC2_21E : MotorControlUDT;
   MCC2_21G : MotorControlUDT;
   MCC2_21K : MotorControlUDT;
   MCC3_2A : MotorControlUDT;
   MCC3_2D : MotorControlUDT;
   MCC3_2G : MotorControlUDT;
   MCC3_2K : MotorControlUDT;
   MCC3_3A : MotorControlUDT;
   MCC3_3D : MotorControlUDT;
   MCC3_3G : MotorControlUDT;
   MCC3_3K : MotorControlUDT;
   MCC3_4A : MotorControlUDT;
   MCC3_4D : MotorControlUDT;
   MCC3_4G : MotorControlUDT;
   MCC3_4K : MotorControlUDT;
   MCC3_5A : MotorControlUDT;
   MCC3_5D : MotorControlUDT;
   MCC3_5G : MotorControlUDT;
   MCC3_5K : MotorControlUDT;
   MCC3_6A : MotorControlUDT;
   MCC3_6D : MotorControlUDT;
   MCC3_6G : MotorControlUDT;
   MCC3_6J : MotorControlUDT;
   MCC3_7A : MotorControlUDT;
   MCC3_7C : MotorControlUDT;
   MCC3_7E : MotorControlUDT;
   MCC3_7G : MotorControlUDT;
   MCC3_7K : MotorControlUDT;
   MCC3_8A : MotorControlUDT;
   MCC3_8D : MotorControlUDT;
   MCC3_8H : MotorControlUDT;
   MCC3_8K : MotorControlUDT;
   MCC3_9A : MotorControlUDT;
   MCC3_9C : MotorControlUDT;
   MCC3_9E : MotorControlUDT;
   MCC3_9G : MotorControlUDT;
   MCC3_9J : MotorControlUDT;
   MCC3_9L : MotorControlUDT;
   MCC3_10A : MotorControlUDT;
   MCC3_10D : MotorControlUDT;
   MCC3_10G : MotorControlUDT;
   MCC3_10J : MotorControlUDT;
   MCC3_11A : MotorControlUDT;
   MCC3_11D : MotorControlUDT;
   MCC3_11G : MotorControlUDT;
   MCC3_11J : MotorControlUDT;
   MCC3_12A : MotorControlUDT;
   MCC3_12C : MotorControlUDT;
   MCC3_12E : MotorControlUDT;
   MCC3_12G : MotorControlUDT;
   MCC3_12J : MotorControlUDT;
   MCC3_12L : MotorControlUDT;
   MCC3_13A : MotorControlUDT;
   MCC3_13C : MotorControlUDT;
   MCC3_13E : MotorControlUDT;
   MCC3_13G : MotorControlUDT;
   MCC3_13J : MotorControlUDT;
   MCC3_13L : MotorControlUDT;
   MCC3_14A : MotorControlUDT;
   MCC3_14C : MotorControlUDT;
   MCC3_14E : MotorControlUDT;
   MCC3_14G : MotorControlUDT;
   MCC3_14J : MotorControlUDT;
   MCC3_14L : MotorControlUDT;
   MCC3_15A : MotorControlUDT;
   MCC3_15C : MotorControlUDT;
   MCC3_15E : MotorControlUDT;
   MCC3_15G : MotorControlUDT;
   MCC3_15J : MotorControlUDT;
   MCC3_16A : MotorControlUDT;
   MCC3_16C : MotorControlUDT;
   MCC3_16E : MotorControlUDT;
   MCC3_16G : MotorControlUDT;
   MCC3_16J : MotorControlUDT;
   MCC3_16L : MotorControlUDT;
   MCC3_17A : MotorControlUDT;
   MCC3_17C : MotorControlUDT;
   MCC3_17E : MotorControlUDT;
   MCC3_17G : MotorControlUDT;
   MCC3_17J : MotorControlUDT;
   MCC3_17L : MotorControlUDT;
   MCC3_18A : MotorControlUDT;
   MCC3_18C : MotorControlUDT;
   MCC3_18E : MotorControlUDT;
   MCC3_18G : MotorControlUDT;
   MCC3_18J : MotorControlUDT;
   MCC3_18L : MotorControlUDT;
   MCC3_19A : MotorControlUDT;
   MCC3_19C : MotorControlUDT;
   MCC3_19E : MotorControlUDT;
   MCC3_19G : MotorControlUDT;
   MCC3_19J : MotorControlUDT;
   MCC3_20A : MotorControlUDT;
   MCC3_20C : MotorControlUDT;
   MCC3_20E : MotorControlUDT;
   MCC3_20G : MotorControlUDT;
   MCC3_20J : MotorControlUDT;
   MCC3_21A : MotorControlUDT;
   MCC3_21C : MotorControlUDT;
   MCC3_21E : MotorControlUDT;
   MCC3_21G : MotorControlUDT;
   MCC3_21J : MotorControlUDT;
   MCC3_21L : MotorControlUDT;
   MCC3_22C : MotorControlUDT;
   MCC3_22E : MotorControlUDT;
   MCC4_1E : MotorControlUDT;
   MCC4_2A : MotorControlUDT;
   MCC4_2C : MotorControlUDT;
   MCC4_2E : MotorControlUDT;
   MCC4_2G : MotorControlUDT;
   MCC4_2K : MotorControlUDT;
   MCC4_3A : MotorControlUDT;
   MCC4_3C : MotorControlUDT;
   MCC4_3E : MotorControlUDT;
   MCC4_3G : MotorControlUDT;
   MCC4_3J : MotorControlUDT;
   MCC4_3L : MotorControlUDT;
   MCC4_4A : MotorControlUDT;
   MCC4_4C : MotorControlUDT;
   MCC4_4E : MotorControlUDT;
   MCC4_4G : MotorControlUDT;
   MCC4_4J : MotorControlUDT;
   MCC4_4L : MotorControlUDT;
   MCC4_5A : MotorControlUDT;
   MCC4_5C : MotorControlUDT;
   MCC4_5E : MotorControlUDT;
   MCC4_5G : MotorControlUDT;
   MCC4_5J : MotorControlUDT;
   MCC4_5L : MotorControlUDT;
END_STRUCT
END_TYPE

TYPE MotorsStatusUDT :   // Structure of All Motor Structures. Status to PLC #1
STRUCT
   MCC2_2A : MotorStatusUDT;
   MCC2_2D : MotorStatusUDT;
   MCC2_2G : MotorStatusUDT;
   MCC2_2K : MotorStatusUDT;
   MCC2_3A : MotorStatusUDT;
   MCC2_3C : MotorStatusUDT;
   MCC2_3E : MotorStatusUDT;
   MCC2_3G : MotorStatusUDT;
   MCC2_3J : MotorStatusUDT;
   MCC2_3L : MotorStatusUDT;
   MCC2_4A : MotorStatusUDT;
   MCC2_4C : MotorStatusUDT;
   MCC2_4E : MotorStatusUDT;
   MCC2_4G : MotorStatusUDT;
   MCC2_4J : MotorStatusUDT;
   MCC2_4L : MotorStatusUDT;
   MCC2_5A : MotorStatusUDT;
   MCC2_5C : MotorStatusUDT;
   MCC2_5E : MotorStatusUDT;
   MCC2_5G : MotorStatusUDT;
   MCC2_5J : MotorStatusUDT;
   MCC2_6A : MotorStatusUDT;
   MCC2_6C : MotorStatusUDT;
   MCC2_6E : MotorStatusUDT;
   MCC2_6G : MotorStatusUDT;
   MCC2_6J : MotorStatusUDT;
   MCC2_6L : MotorStatusUDT;
   MCC2_7A : MotorStatusUDT;
   MCC2_7D : MotorStatusUDT;
   MCC2_7G : MotorStatusUDT;
   MCC2_7K : MotorStatusUDT;
   MCC2_8B : MotorStatusUDT;
   MCC2_8D : MotorStatusUDT;
   MCC2_8F : MotorStatusUDT;
   MCC2_8H : MotorStatusUDT;
   MCC2_8K : MotorStatusUDT;
   MCC2_9D : MotorStatusUDT;
   MCC2_9F : MotorStatusUDT;
   MCC2_9H : MotorStatusUDT;
   MCC2_10A : MotorStatusUDT;
   MCC2_10C : MotorStatusUDT;
   MCC2_10E : MotorStatusUDT;
   MCC2_10G : MotorStatusUDT;
   MCC2_10J : MotorStatusUDT;
   MCC2_10L : MotorStatusUDT;
   MCC2_11A : MotorStatusUDT;
   MCC2_11C : MotorStatusUDT;
   MCC2_11E : MotorStatusUDT;
   MCC2_11G : MotorStatusUDT;
   MCC2_11J : MotorStatusUDT;
   MCC2_11L : MotorStatusUDT;
   MCC2_12A : MotorStatusUDT;
   MCC2_12C : MotorStatusUDT;
   MCC2_12E : MotorStatusUDT;
   MCC2_12G : MotorStatusUDT;
   MCC2_12J : MotorStatusUDT;
   MCC2_12L : MotorStatusUDT;
   MCC2_13A : MotorStatusUDT;
   MCC2_13C : MotorStatusUDT;
   MCC2_13E : MotorStatusUDT;
   MCC2_13G : MotorStatusUDT;
   MCC2_13J : MotorStatusUDT;
   MCC2_14A : MotorStatusUDT;
   MCC2_14C : MotorStatusUDT;
   MCC2_14E : MotorStatusUDT;
   MCC2_14G : MotorStatusUDT;
   MCC2_14J : MotorStatusUDT;
   MCC2_14L : MotorStatusUDT;
   MCC2_15A : MotorStatusUDT;
   MCC2_15C : MotorStatusUDT;
   MCC2_15E : MotorStatusUDT;
   MCC2_15G : MotorStatusUDT;
   MCC2_15J : MotorStatusUDT;
   MCC2_15L : MotorStatusUDT;
   MCC2_16A : MotorStatusUDT;
   MCC2_16C : MotorStatusUDT;
   MCC2_16E : MotorStatusUDT;
   MCC2_16G : MotorStatusUDT;
   MCC2_16J : MotorStatusUDT;
   MCC2_16L : MotorStatusUDT;
   MCC2_17A : MotorStatusUDT;
   MCC2_17C : MotorStatusUDT;
   MCC2_17E : MotorStatusUDT;
   MCC2_17G : MotorStatusUDT;
   MCC2_17J : MotorStatusUDT;
   MCC2_18A : MotorStatusUDT;
   MCC2_18C : MotorStatusUDT;
   MCC2_18E : MotorStatusUDT;
   MCC2_18G : MotorStatusUDT;
   MCC2_18J : MotorStatusUDT;
   MCC2_18L : MotorStatusUDT;
   MCC2_19A : MotorStatusUDT;
   MCC2_19C : MotorStatusUDT;
   MCC2_19E : MotorStatusUDT;
   MCC2_19G : MotorStatusUDT;
   MCC2_19J : MotorStatusUDT;
   MCC2_19L : MotorStatusUDT;
   MCC2_20C : MotorStatusUDT;
   MCC2_20E : MotorStatusUDT;
   MCC2_20G : MotorStatusUDT;
   MCC2_20J : MotorStatusUDT;
   MCC2_21A : MotorStatusUDT;
   MCC2_21C : MotorStatusUDT;
   MCC2_21E : MotorStatusUDT;
   MCC2_21G : MotorStatusUDT;
   MCC2_21K : MotorStatusUDT;
   MCC3_2A : MotorStatusUDT;
   MCC3_2D : MotorStatusUDT;
   MCC3_2G : MotorStatusUDT;
   MCC3_2K : MotorStatusUDT;
   MCC3_3A : MotorStatusUDT;
   MCC3_3D : MotorStatusUDT;
   MCC3_3G : MotorStatusUDT;
   MCC3_3K : MotorStatusUDT;
   MCC3_4A : MotorStatusUDT;
   MCC3_4D : MotorStatusUDT;
   MCC3_4G : MotorStatusUDT;
   MCC3_4K : MotorStatusUDT;
   MCC3_5A : MotorStatusUDT;
   MCC3_5D : MotorStatusUDT;
   MCC3_5G : MotorStatusUDT;
   MCC3_5K : MotorStatusUDT;
   MCC3_6A : MotorStatusUDT;
   MCC3_6D : MotorStatusUDT;
   MCC3_6G : MotorStatusUDT;
   MCC3_6J : MotorStatusUDT;
   MCC3_7A : MotorStatusUDT;
   MCC3_7C : MotorStatusUDT;
   MCC3_7E : MotorStatusUDT;
   MCC3_7G : MotorStatusUDT;
   MCC3_7K : MotorStatusUDT;
   MCC3_8A : MotorStatusUDT;
   MCC3_8D : MotorStatusUDT;
   MCC3_8H : MotorStatusUDT;
   MCC3_8K : MotorStatusUDT;
   MCC3_9A : MotorStatusUDT;
   MCC3_9C : MotorStatusUDT;
   MCC3_9E : MotorStatusUDT;
   MCC3_9G : MotorStatusUDT;
   MCC3_9J : MotorStatusUDT;
   MCC3_9L : MotorStatusUDT;
   MCC3_10A : MotorStatusUDT;
   MCC3_10D : MotorStatusUDT;
   MCC3_10G : MotorStatusUDT;
   MCC3_10J : MotorStatusUDT;
   MCC3_11A : MotorStatusUDT;
   MCC3_11D : MotorStatusUDT;
   MCC3_11G : MotorStatusUDT;
   MCC3_11J : MotorStatusUDT;
   MCC3_12A : MotorStatusUDT;
   MCC3_12C : MotorStatusUDT;
   MCC3_12E : MotorStatusUDT;
   MCC3_12G : MotorStatusUDT;
   MCC3_12J : MotorStatusUDT;
   MCC3_12L : MotorStatusUDT;
   MCC3_13A : MotorStatusUDT;
   MCC3_13C : MotorStatusUDT;
   MCC3_13E : MotorStatusUDT;
   MCC3_13G : MotorStatusUDT;
   MCC3_13J : MotorStatusUDT;
   MCC3_13L : MotorStatusUDT;
   MCC3_14A : MotorStatusUDT;
   MCC3_14C : MotorStatusUDT;
   MCC3_14E : MotorStatusUDT;
   MCC3_14G : MotorStatusUDT;
   MCC3_14J : MotorStatusUDT;
   MCC3_14L : MotorStatusUDT;
   MCC3_15A : MotorStatusUDT;
   MCC3_15C : MotorStatusUDT;
   MCC3_15E : MotorStatusUDT;
   MCC3_15G : MotorStatusUDT;
   MCC3_15J : MotorStatusUDT;
   MCC3_16A : MotorStatusUDT;
   MCC3_16C : MotorStatusUDT;
   MCC3_16E : MotorStatusUDT;
   MCC3_16G : MotorStatusUDT;
   MCC3_16J : MotorStatusUDT;
   MCC3_16L : MotorStatusUDT;
   MCC3_17A : MotorStatusUDT;
   MCC3_17C : MotorStatusUDT;
   MCC3_17E : MotorStatusUDT;
   MCC3_17G : MotorStatusUDT;
   MCC3_17J : MotorStatusUDT;
   MCC3_17L : MotorStatusUDT;
   MCC3_18A : MotorStatusUDT;
   MCC3_18C : MotorStatusUDT;
   MCC3_18E : MotorStatusUDT;
   MCC3_18G : MotorStatusUDT;
   MCC3_18J : MotorStatusUDT;
   MCC3_18L : MotorStatusUDT;
   MCC3_19A : MotorStatusUDT;
   MCC3_19C : MotorStatusUDT;
   MCC3_19E : MotorStatusUDT;
   MCC3_19G : MotorStatusUDT;
   MCC3_19J : MotorStatusUDT;
   MCC3_20A : MotorStatusUDT;
   MCC3_20C : MotorStatusUDT;
   MCC3_20E : MotorStatusUDT;
   MCC3_20G : MotorStatusUDT;
   MCC3_20J : MotorStatusUDT;
   MCC3_21A : MotorStatusUDT;
   MCC3_21C : MotorStatusUDT;
   MCC3_21E : MotorStatusUDT;
   MCC3_21G : MotorStatusUDT;
   MCC3_21J : MotorStatusUDT;
   MCC3_21L : MotorStatusUDT;
   MCC3_22C : MotorStatusUDT;
   MCC3_22E : MotorStatusUDT;
   MCC4_1E : MotorStatusUDT;
   MCC4_2A : MotorStatusUDT;
   MCC4_2C : MotorStatusUDT;
   MCC4_2E : MotorStatusUDT;
   MCC4_2G : MotorStatusUDT;
   MCC4_2K : MotorStatusUDT;
   MCC4_3A : MotorStatusUDT;
   MCC4_3C : MotorStatusUDT;
   MCC4_3E : MotorStatusUDT;
   MCC4_3G : MotorStatusUDT;
   MCC4_3J : MotorStatusUDT;
   MCC4_3L : MotorStatusUDT;
   MCC4_4A : MotorStatusUDT;
   MCC4_4C : MotorStatusUDT;
   MCC4_4E : MotorStatusUDT;
   MCC4_4G : MotorStatusUDT;
   MCC4_4J : MotorStatusUDT;
   MCC4_4L : MotorStatusUDT;
   MCC4_5A : MotorStatusUDT;
   MCC4_5C : MotorStatusUDT;
   MCC4_5E : MotorStatusUDT;
   MCC4_5G : MotorStatusUDT;
   MCC4_5J : MotorStatusUDT;
   MCC4_5L : MotorStatusUDT;
END_STRUCT
END_TYPE

TYPE MotorStatusUDT :   // Motor Status to PLC #1
STRUCT
   StatusBits : DINT;   // Status Bits
   Amps : REAL;   // Motor Amps
   OverloadPercent : DINT;   // Motor Overload 0->100%
   MSG_FaultWarning : DINT;   // Fault / Warning Message to PLC1
   Spare : DINT;   // Spare DINT Element
END_STRUCT
END_TYPE

ADD_ON_INSTRUCTION E300ToMotor   (* revision 1.0 *)
// Get Information from E300 AOP Input to Motor UTD
VAR_IN_OUT
   MotorTemp : MotorStatusUDT; {required}   // Motor UDT Temporary
        .StatusBits   // Status Bits..0=Running, 1 = Warning, 2=Fault
   AOP_E300_I_Temp : AB:E300:I:3; {required}   // Input Data from E300 AOP Inputs
END_VAR
VAR_INPUT
   CommsOK : BOOL; {required}   // Communications OK
END_VAR

ROUTINE Logic   (* ladder *)
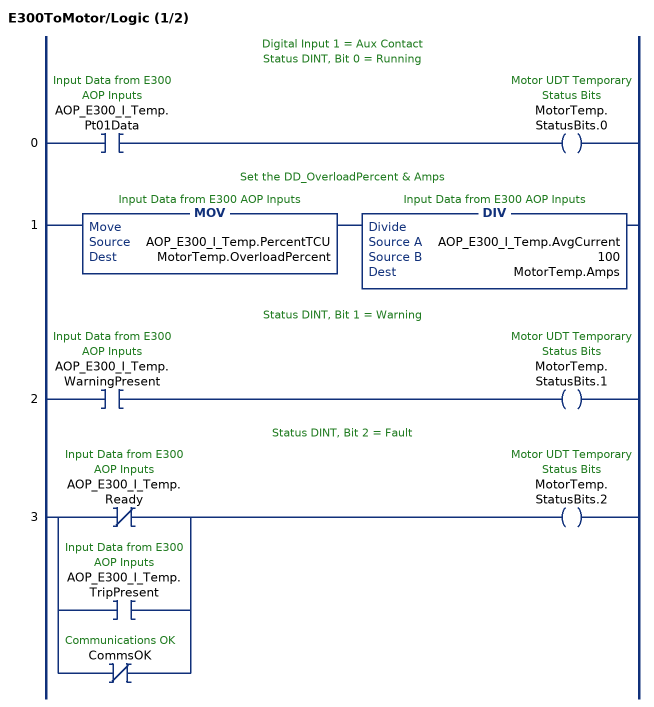
   // Digital Input 1 = Aux Contact
   // Status DINT, Bit 0 = Running
   0: XIC(AOP_E300_I_Temp.Pt01Data)OTE(MotorTemp.StatusBits.0);
   // Set the DD_OverloadPercent & Amps
   1: MOV(AOP_E300_I_Temp.PercentTCU,MotorTemp.OverloadPercent)DIV(AOP_E300_I_Temp.AvgCurrent,100,MotorTemp.Amps);
   // Status DINT, Bit 1 = Warning
   2: XIC(AOP_E300_I_Temp.WarningPresent)OTE(MotorTemp.StatusBits.1);
   // Status DINT, Bit 2 = Fault
   3: [XIO(AOP_E300_I_Temp.Ready) ,XIC(AOP_E300_I_Temp.TripPresent) ,XIO(CommsOK) ]OTE(MotorTemp.StatusBits.2);
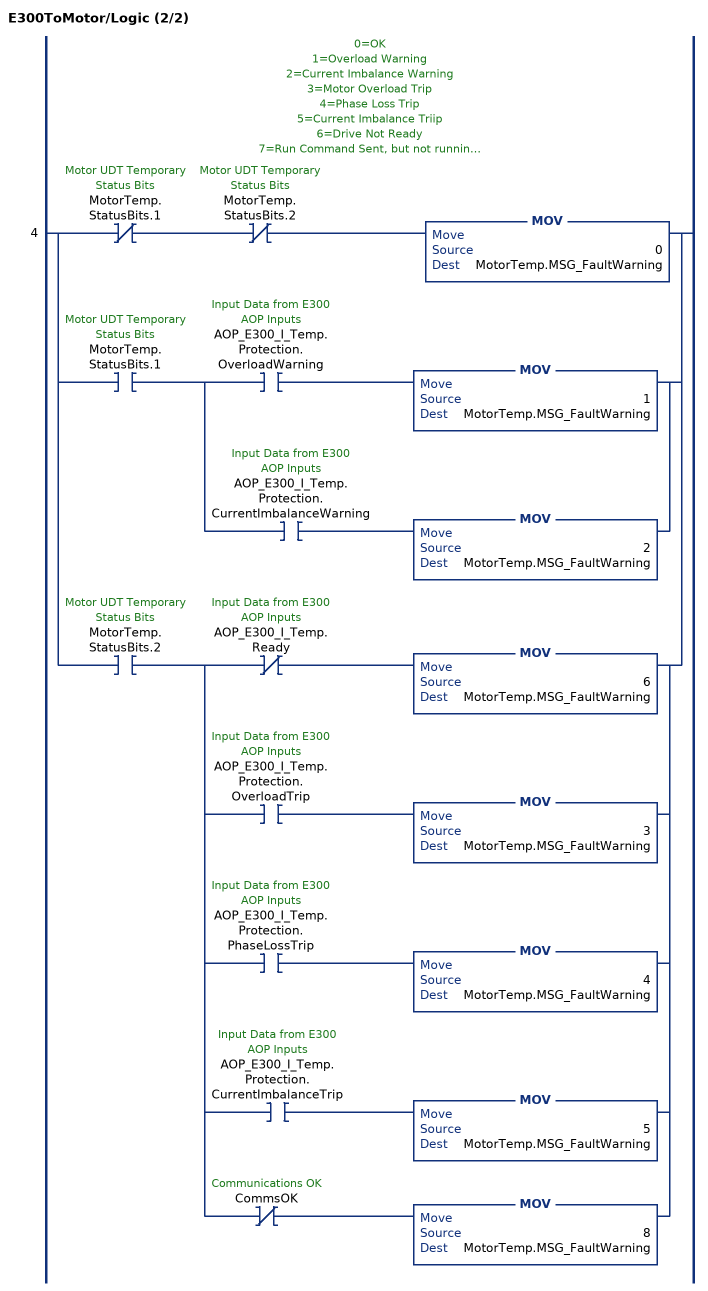
   // 0=OK
   // 1=Overload Warning
   // 2=Current Imbalance Warning
   // 3=Motor Overload Trip
   // 4=Phase Loss Trip
   // 5=Current Imbalance Triip
   // 6=Drive Not Ready
   // 7=Run Command Sent, but not running
   // 8=Loss Of Ethernet Communications
   // 9=VFD Fault
   // 10=Motion Alarm
   4: [XIO(MotorTemp.StatusBits.1) XIO(MotorTemp.StatusBits.2) MOV(0,MotorTemp.MSG_FaultWarning) ,[XIC(MotorTemp.StatusBits.1) [XIC(AOP_E300_I_Temp.Protection.OverloadWarning) MOV(1,MotorTemp.MSG_FaultWarning) ,XIC(AOP_E300_I_Temp.Protection.CurrentImbalanceWarning) MOV(2,MotorTemp.MSG_FaultWarning) ] ,XIC(MotorTemp.StatusBits.2) [XIO(AOP_E300_I_Temp.Ready) MOV(6,MotorTemp.MSG_FaultWarning) ,XIC(AOP_E300_I_Temp.Protection.OverloadTrip) MOV(3,MotorTemp.MSG_FaultWarning) ,XIC(AOP_E300_I_Temp.Protection.PhaseLossTrip) MOV(4,MotorTemp.MSG_FaultWarning) ,XIC(AOP_E300_I_Temp.Protection.CurrentImbalanceTrip) MOV(5,MotorTemp.MSG_FaultWarning) ,XIO(CommsOK) MOV(8,MotorTemp.MSG_FaultWarning) ] ] ];
END_ROUTINE
END_ADD_ON_INSTRUCTION

ADD_ON_INSTRUCTION MotorToE300   (* revision 1.0 *)
// Motor UDT Output to E300
VAR_IN_OUT
   AOP_E300_O_Temp : AB:E300:O:1; {required}   // Output Data to E300 AOP
   MotorTemp : MotorControlUDT; {required}   // MotorFromPLC1 UDT to send to E300
END_VAR
VAR_INPUT
   OK : BOOL; {required}   // OK To Run
END_VAR

ROUTINE Logic   (* ladder *)
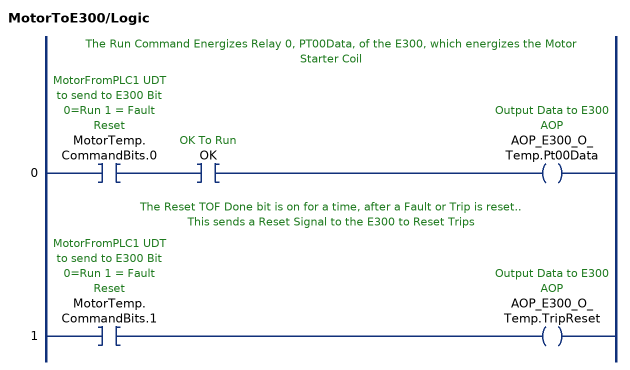
   // The Run Command Energizes Relay 0, PT00Data, of the E300, which energizes the Motor Starter Coil
   0: XIC(MotorTemp.CommandBits.0)XIC(OK)OTE(AOP_E300_O_Temp.Pt00Data);
   // The Reset TOF Done bit is on for a time, after a Fault or Trip is reset..
   // This sends a Reset Signal to the E300 to Reset Trips
   1: XIC(MotorTemp.CommandBits.1)OTE(AOP_E300_O_Temp.TripReset);
END_ROUTINE
END_ADD_ON_INSTRUCTION

ADD_ON_INSTRUCTION MotorToPF525   (* revision 1.0 *)
// Motor UDT to PF525 Commands & Speed
VAR_IN_OUT
   AOP_PF525_O_Temp : AB:PowerFlex525V_EENET_Drive:O:0; {required}   // PF525 AOP Output Data
   MotorTemp : MotorControlUDT; {required}   // Motor UDT to PF525 Commands Bit0=Run, 1=Fault Reset
END_VAR
VAR_INPUT
   OK : BOOL; {access None, required}   // Ok To Run
END_VAR
VAR
   StopPulseTimer : TIMER := (PRE := 1500); {access None}
END_VAR

ROUTINE Logic   (* ladder *)
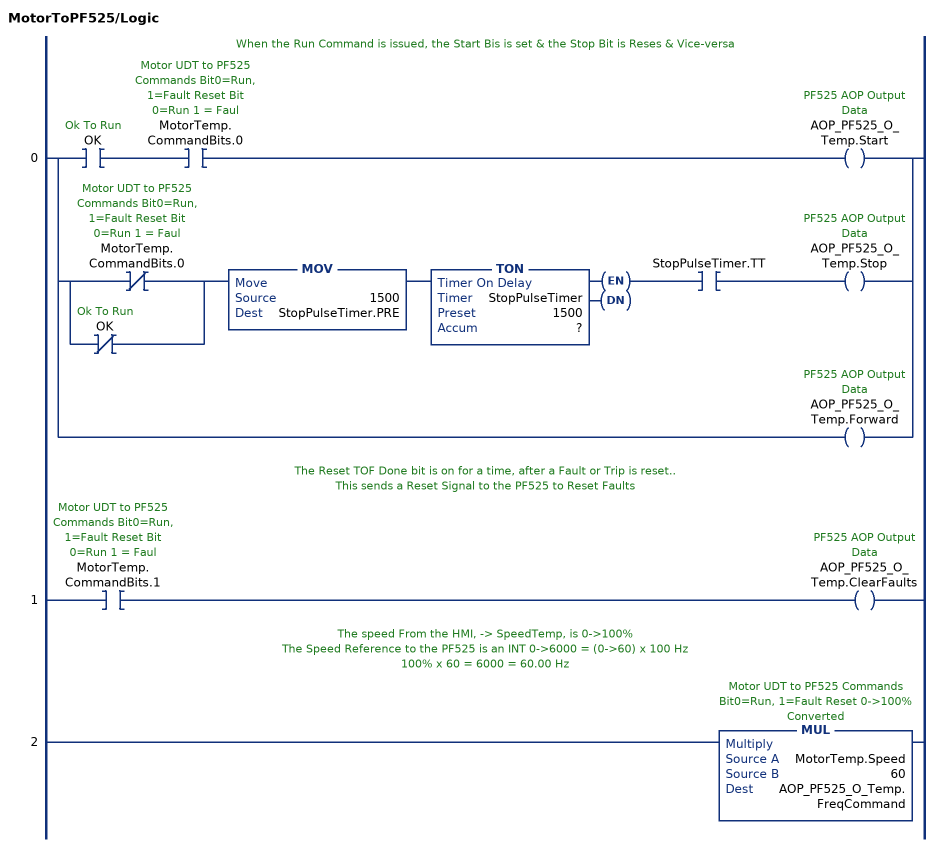
   // When the Run Command is issued, the Start Bis is set & the Stop Bit is Reses & Vice-versa
   0: [XIC(OK) XIC(MotorTemp.CommandBits.0) OTE(AOP_PF525_O_Temp.Start) ,[XIO(MotorTemp.CommandBits.0) ,XIO(OK) ] MOV(1500,StopPulseTimer.PRE) TON(StopPulseTimer,?,?) XIC(StopPulseTimer.TT) OTE(AOP_PF525_O_Temp.Stop) ,OTE(AOP_PF525_O_Temp.Forward) ];
   // The Reset TOF Done bit is on for a time, after a Fault or Trip is reset..
   // This sends a Reset Signal to the PF525 to Reset Faults
   1: XIC(MotorTemp.CommandBits.1)OTE(AOP_PF525_O_Temp.ClearFaults);
   // The speed From the HMI, -> SpeedTemp, is 0->100%
   // The Speed Reference to the PF525 is an INT 0->6000 = (0->60) x 100 Hz
   // 100% x 60 = 6000 = 60.00 Hz
   2: MUL(MotorTemp.Speed,60,AOP_PF525_O_Temp.FreqCommand);
END_ROUTINE
END_ADD_ON_INSTRUCTION

ADD_ON_INSTRUCTION PF525ToMotor   (* revision 1.0 *)
// Get PF525 AOP Input Data to Motor UDT & Update Motor Status
VAR_IN_OUT
   MotorTemp : MotorStatusUDT; {required}   // Motor UDT Temporary
        .StatusBits   // Status Bits to PC#1: 0=Running, 1=Warning, 2=Fault
   PF525_AOP_I_Temp : AB:PowerFlex525V_E_1A80B093:I:0; {required}   // Input Data from PF525 AOP Inputs
END_VAR
VAR_INPUT
   CommsOK : BOOL; {required}   // AOP Communications OK
END_VAR

ROUTINE Logic   (* ladder *)
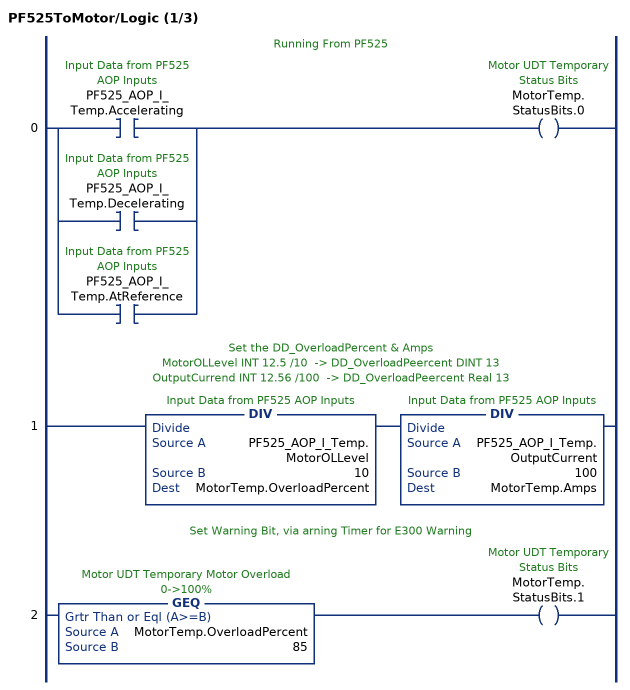
   // Running From PF525
   0: [XIC(PF525_AOP_I_Temp.Accelerating) ,XIC(PF525_AOP_I_Temp.Decelerating) ,XIC(PF525_AOP_I_Temp.AtReference) ]OTE(MotorTemp.StatusBits.0);
   // Set the DD_OverloadPercent & Amps
   // MotorOLLevel INT 12.5 /10  -> DD_OverloadPeercent DINT 13
   // OutputCurrend INT 12.56 /100  -> DD_OverloadPeercent Real 13
   1: DIV(PF525_AOP_I_Temp.MotorOLLevel,10,MotorTemp.OverloadPercent)DIV(PF525_AOP_I_Temp.OutputCurrent,100,MotorTemp.Amps);
   // Set Warning Bit, via arning Timer for E300 Warning
   2: GEQ(MotorTemp.OverloadPercent,85)OTE(MotorTemp.StatusBits.1);
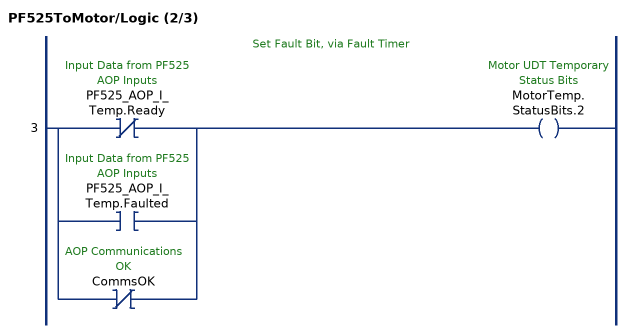
   // Set Fault Bit, via Fault Timer
   3: [XIO(PF525_AOP_I_Temp.Ready) ,XIC(PF525_AOP_I_Temp.Faulted) ,XIO(CommsOK) ]OTE(MotorTemp.StatusBits.2);
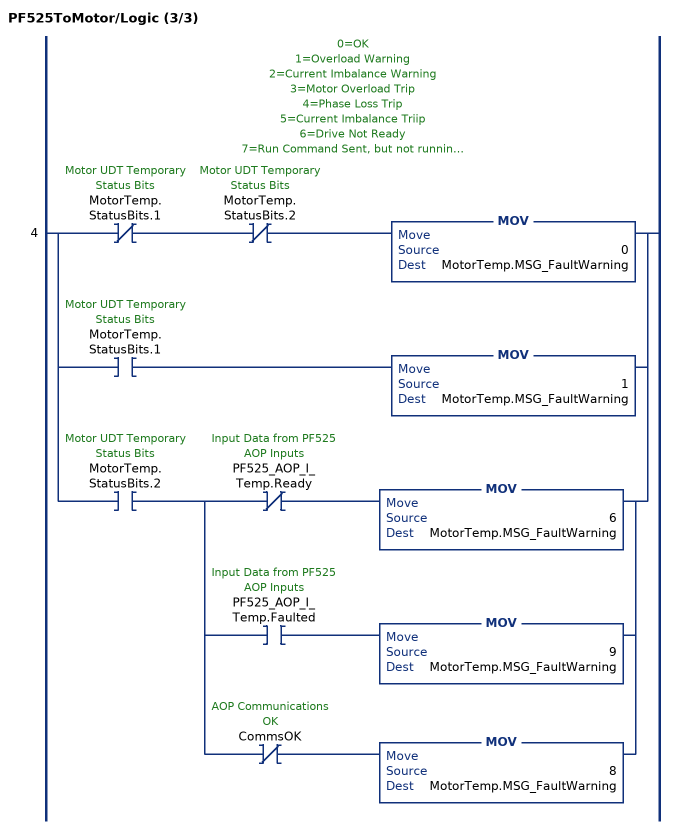
   // 0=OK
   // 1=Overload Warning
   // 2=Current Imbalance Warning
   // 3=Motor Overload Trip
   // 4=Phase Loss Trip
   // 5=Current Imbalance Triip
   // 6=Drive Not Ready
   // 7=Run Command Sent, but not running
   // 8=Loss Of Ethernet Communications
   // 9=VFD Fault
   // 10=Motion Alarm
   4: [XIO(MotorTemp.StatusBits.1) XIO(MotorTemp.StatusBits.2) MOV(0,MotorTemp.MSG_FaultWarning) ,[XIC(MotorTemp.StatusBits.1) MOV(1,MotorTemp.MSG_FaultWarning) ,XIC(MotorTemp.StatusBits.2) [XIO(PF525_AOP_I_Temp.Ready) MOV(6,MotorTemp.MSG_FaultWarning) ,XIC(PF525_AOP_I_Temp.Faulted) MOV(9,MotorTemp.MSG_FaultWarning) ,XIO(CommsOK) MOV(8,MotorTemp.MSG_FaultWarning) ] ] ];
END_ROUTINE
END_ADD_ON_INSTRUCTION

VAR_GLOBAL   (* controller tags *)
   AFI : BOOL;   // Always False
   AOI_MCC2_10A_ToPLC1 : E300ToMotor := (CommsOK := 1);
   AOI_MCC2_10C_ToPLC1 : E300ToMotor := (CommsOK := 1);
   AOI_MCC2_10E_ToPLC1 : E300ToMotor := (CommsOK := 1);
   AOI_MCC2_10G_ToPLC1 : E300ToMotor := (CommsOK := 1);
   AOI_MCC2_10J_ToPLC1 : E300ToMotor := (CommsOK := 1);
   AOI_MCC2_10L_ToPLC1 : E300ToMotor := (CommsOK := 1);
   AOI_MCC2_11A_ToPLC1 : E300ToMotor := (CommsOK := 1);
   AOI_MCC2_11C_ToPLC1 : E300ToMotor := (CommsOK := 1);
   AOI_MCC2_11E_ToPLC1 : E300ToMotor := (CommsOK := 1);
   AOI_MCC2_11G_ToPLC1 : E300ToMotor := (CommsOK := 1);
   AOI_MCC2_11J_ToPLC1 : E300ToMotor := (CommsOK := 1);
   AOI_MCC2_11L_ToPLC1 : E300ToMotor;
   AOI_MCC2_12A_ToPLC1 : E300ToMotor := (CommsOK := 1);
   AOI_MCC2_12C_ToPLC1 : E300ToMotor := (CommsOK := 1);
   AOI_MCC2_12E_ToPLC1 : E300ToMotor := (CommsOK := 1);
   AOI_MCC2_12G_ToPLC1 : E300ToMotor := (CommsOK := 1);
   AOI_MCC2_12J_ToPLC1 : E300ToMotor := (CommsOK := 1);
   AOI_MCC2_12L_ToPLC1 : E300ToMotor := (CommsOK := 1);
   AOI_MCC2_13A_ToPLC1 : E300ToMotor := (CommsOK := 1);
   AOI_MCC2_13C_ToPLC1 : E300ToMotor := (CommsOK := 1);
   AOI_MCC2_13E_ToPLC1 : E300ToMotor;
   AOI_MCC2_13G_ToPLC1 : E300ToMotor := (CommsOK := 1);
   AOI_MCC2_13J_ToPLC1 : E300ToMotor := (CommsOK := 1);
   AOI_MCC2_14A_ToPLC1 : E300ToMotor := (CommsOK := 1);
   AOI_MCC2_14C_ToPLC1 : E300ToMotor := (CommsOK := 1);
   AOI_MCC2_14E_ToPLC1 : E300ToMotor := (CommsOK := 1);
   AOI_MCC2_14G_ToPLC1 : E300ToMotor := (CommsOK := 1);
   AOI_MCC2_14J_ToPLC1 : E300ToMotor;
   AOI_MCC2_14L_ToPLC1 : E300ToMotor := (CommsOK := 1);
   AOI_MCC2_15A_ToPLC1 : E300ToMotor := (CommsOK := 1);
   AOI_MCC2_15C_ToPLC1 : E300ToMotor := (CommsOK := 1);
   AOI_MCC2_15E_ToPLC1 : E300ToMotor := (CommsOK := 1);
   AOI_MCC2_15G_ToPLC1 : E300ToMotor := (CommsOK := 1);
   AOI_MCC2_15J_ToPLC1 : E300ToMotor := (CommsOK := 1);
   AOI_MCC2_15L_ToPLC1 : E300ToMotor := (CommsOK := 1);
   AOI_MCC2_16A_ToPLC1 : E300ToMotor := (CommsOK := 1);
   AOI_MCC2_16C_ToPLC1 : E300ToMotor := (CommsOK := 1);
   AOI_MCC2_16E_ToPLC1 : E300ToMotor := (CommsOK := 1);
   AOI_MCC2_16G_ToPLC1 : E300ToMotor := (CommsOK := 1);
   AOI_MCC2_16J_ToPLC1 : E300ToMotor := (CommsOK := 1);
   AOI_MCC2_16L_ToPLC1 : E300ToMotor := (CommsOK := 1);
   AOI_MCC2_17A_ToPLC1 : E300ToMotor := (CommsOK := 1);
   AOI_MCC2_17C_ToPLC1 : E300ToMotor := (CommsOK := 1);
   AOI_MCC2_17E_ToPLC1 : E300ToMotor := (CommsOK := 1);
   AOI_MCC2_17G_ToPLC1 : E300ToMotor := (CommsOK := 1);
   AOI_MCC2_17J_ToPLC1 : E300ToMotor := (CommsOK := 1);
   AOI_MCC2_18A_ToPLC1 : E300ToMotor := (CommsOK := 1);
   AOI_MCC2_18C_ToPLC1 : E300ToMotor := (CommsOK := 1);
   AOI_MCC2_18E_ToPLC1 : E300ToMotor := (CommsOK := 1);
   AOI_MCC2_18G_ToPLC1 : E300ToMotor := (CommsOK := 1);
   AOI_MCC2_18J_ToPLC1 : E300ToMotor := (CommsOK := 1);
   AOI_MCC2_18L_ToPLC1 : E300ToMotor := (CommsOK := 1);
   AOI_MCC2_19A_ToPLC1 : E300ToMotor := (CommsOK := 1);
   AOI_MCC2_19C_ToPLC1 : E300ToMotor := (CommsOK := 1);
   AOI_MCC2_19E_ToPLC1 : E300ToMotor := (CommsOK := 1);
   AOI_MCC2_19G_ToPLC1 : E300ToMotor := (CommsOK := 1);
   AOI_MCC2_19J_ToPLC1 : E300ToMotor := (CommsOK := 1);
   AOI_MCC2_19L_ToPLC1 : E300ToMotor := (CommsOK := 1);
   AOI_MCC2_20C_ToPLC1 : E300ToMotor := (CommsOK := 1);
   AOI_MCC2_20E_ToPLC1 : E300ToMotor := (CommsOK := 1);
   AOI_MCC2_20G_ToPLC1 : E300ToMotor;
   AOI_MCC2_20J_ToPLC1 : E300ToMotor := (CommsOK := 1);
   AOI_MCC2_21A_ToPLC1 : E300ToMotor := (CommsOK := 1);
   AOI_MCC2_21C_ToPLC1 : E300ToMotor := (CommsOK := 1);
   AOI_MCC2_21E_ToPLC1 : E300ToMotor := (CommsOK := 1);
   AOI_MCC2_21G_ToPLC1 : PF525ToMotor := (CommsOK := 1);
   AOI_MCC2_21K_ToPLC1 : PF525ToMotor;
   AOI_MCC2_2A_ToPLC1 : PF525ToMotor := (CommsOK := 1);
   AOI_MCC2_2D_ToPLC1 : PF525ToMotor := (CommsOK := 1);
   AOI_MCC2_2G_ToPLC1 : PF525ToMotor := (CommsOK := 1);
   AOI_MCC2_2K_ToPLC1 : PF525ToMotor := (CommsOK := 1);
   AOI_MCC2_3A_ToPLC1 : E300ToMotor := (CommsOK := 1);
   AOI_MCC2_3C_ToPLC1 : E300ToMotor := (CommsOK := 1);
   AOI_MCC2_3E_ToPLC1 : E300ToMotor := (CommsOK := 1);
   AOI_MCC2_3G_ToPLC1 : E300ToMotor := (CommsOK := 1);
   AOI_MCC2_3J_ToPLC1 : E300ToMotor := (CommsOK := 1);
   AOI_MCC2_3L_ToPLC1 : E300ToMotor := (CommsOK := 1);
   AOI_MCC2_4A_ToPLC1 : E300ToMotor := (CommsOK := 1);
   AOI_MCC2_4C_ToPLC1 : E300ToMotor := (CommsOK := 1);
   AOI_MCC2_4E_ToPLC1 : E300ToMotor := (CommsOK := 1);
   AOI_MCC2_4G_ToPLC1 : E300ToMotor := (CommsOK := 1);
   AOI_MCC2_4J_ToPLC1 : E300ToMotor := (CommsOK := 1);
   AOI_MCC2_4L_ToPLC1 : E300ToMotor := (CommsOK := 1);
   AOI_MCC2_5A_ToPLC1 : E300ToMotor := (CommsOK := 1);
   AOI_MCC2_5C_ToPLC1 : E300ToMotor := (CommsOK := 1);
   AOI_MCC2_5E_ToPLC1 : E300ToMotor := (CommsOK := 1);
   AOI_MCC2_5G_ToPLC1 : E300ToMotor := (CommsOK := 1);
   AOI_MCC2_5J_ToPLC1 : E300ToMotor := (CommsOK := 1);
   AOI_MCC2_6A_ToPLC1 : E300ToMotor := (CommsOK := 1);
   AOI_MCC2_6C_ToPLC1 : E300ToMotor := (CommsOK := 1);
   AOI_MCC2_6E_ToPLC1 : E300ToMotor := (CommsOK := 1);
   AOI_MCC2_6G_ToPLC1 : E300ToMotor := (CommsOK := 1);
   AOI_MCC2_6J_ToPLC1 : E300ToMotor := (CommsOK := 1);
   AOI_MCC2_6L_ToPLC1 : E300ToMotor := (CommsOK := 1);
   AOI_MCC2_7A_ToPLC1 : E300ToMotor := (CommsOK := 1);
   AOI_MCC2_7D_ToPLC1 : E300ToMotor := (CommsOK := 1);
   AOI_MCC2_7G_ToPLC1 : E300ToMotor := (CommsOK := 1);
   AOI_MCC2_7K_ToPLC1 : E300ToMotor;
   AOI_MCC2_8B_ToPLC1 : E300ToMotor;
   AOI_MCC2_8D_ToPLC1 : E300ToMotor := (CommsOK := 1);
   AOI_MCC2_8F_ToPLC1 : E300ToMotor := (CommsOK := 1);
   AOI_MCC2_8H_ToPLC1 : E300ToMotor := (CommsOK := 1);
   AOI_MCC2_8K_ToPLC1 : E300ToMotor;
   AOI_MCC2_9D_ToPLC1 : E300ToMotor := (CommsOK := 1);
   AOI_MCC2_9F_ToPLC1 : E300ToMotor := (CommsOK := 1);
   AOI_MCC2_9H_ToPLC1 : PF525ToMotor := (CommsOK := 1);
   AOI_MCC3_10A_ToPLC1 : E300ToMotor := (CommsOK := 1);
   AOI_MCC3_10D_ToPLC1 : E300ToMotor;
   AOI_MCC3_10G_ToPLC1 : E300ToMotor := (CommsOK := 1);
   AOI_MCC3_10J_ToPLC1 : E300ToMotor;
   AOI_MCC3_11A_ToPLC1 : E300ToMotor := (CommsOK := 1);
   AOI_MCC3_11D_ToPLC1 : E300ToMotor := (CommsOK := 1);
   AOI_MCC3_11G_ToPLC1 : E300ToMotor := (CommsOK := 1);
   AOI_MCC3_11J_ToPLC1 : E300ToMotor;
   AOI_MCC3_12A_ToPLC1 : E300ToMotor;
   AOI_MCC3_12C_ToPLC1 : E300ToMotor := (CommsOK := 1);
   AOI_MCC3_12E_ToPLC1 : E300ToMotor := (CommsOK := 1);
   AOI_MCC3_12G_ToPLC1 : E300ToMotor := (CommsOK := 1);
   AOI_MCC3_12J_ToPLC1 : E300ToMotor := (CommsOK := 1);
   AOI_MCC3_12L_ToPLC1 : E300ToMotor := (CommsOK := 1);
   AOI_MCC3_13A_ToPLC1 : E300ToMotor := (CommsOK := 1);
   AOI_MCC3_13C_ToPLC1 : E300ToMotor := (CommsOK := 1);
   AOI_MCC3_13E_ToPLC1 : E300ToMotor := (CommsOK := 1);
   AOI_MCC3_13G_ToPLC1 : E300ToMotor := (CommsOK := 1);
   AOI_MCC3_13J_ToPLC1 : E300ToMotor := (CommsOK := 1);
   AOI_MCC3_13L_ToPLC1 : E300ToMotor := (CommsOK := 1);
   AOI_MCC3_14A_ToPLC1 : E300ToMotor := (CommsOK := 1);
   AOI_MCC3_14C_ToPLC1 : E300ToMotor := (CommsOK := 1);
   AOI_MCC3_14E_ToPLC1 : E300ToMotor := (CommsOK := 1);
   AOI_MCC3_14G_ToPLC1 : E300ToMotor := (CommsOK := 1);
   AOI_MCC3_14J_ToPLC1 : E300ToMotor := (CommsOK := 1);
   AOI_MCC3_14L_ToPLC1 : E300ToMotor;
   AOI_MCC3_15A_ToPLC1 : E300ToMotor := (CommsOK := 1);
   AOI_MCC3_15C_ToPLC1 : E300ToMotor := (CommsOK := 1);
   AOI_MCC3_15E_ToPLC1 : E300ToMotor := (CommsOK := 1);
   AOI_MCC3_15G_ToPLC1 : E300ToMotor := (CommsOK := 1);
   AOI_MCC3_15J_ToPLC1 : E300ToMotor;
   AOI_MCC3_16A_ToPLC1 : E300ToMotor := (CommsOK := 1);
   AOI_MCC3_16C_ToPLC1 : E300ToMotor := (CommsOK := 1);
   AOI_MCC3_16E_ToPLC1 : E300ToMotor;
   AOI_MCC3_16G_ToPLC1 : E300ToMotor := (CommsOK := 1);
   AOI_MCC3_16J_ToPLC1 : E300ToMotor := (CommsOK := 1);
   AOI_MCC3_16L_ToPLC1 : E300ToMotor := (CommsOK := 1);
   AOI_MCC3_17A_ToPLC1 : E300ToMotor := (CommsOK := 1);
   AOI_MCC3_17C_ToPLC1 : E300ToMotor := (CommsOK := 1);
   AOI_MCC3_17E_ToPLC1 : E300ToMotor := (CommsOK := 1);
   AOI_MCC3_17G_ToPLC1 : E300ToMotor := (CommsOK := 1);
   AOI_MCC3_17J_ToPLC1 : E300ToMotor := (CommsOK := 1);
   AOI_MCC3_17L_ToPLC1 : E300ToMotor := (CommsOK := 1);
   AOI_MCC3_18A_ToPLC1 : E300ToMotor := (CommsOK := 1);
   AOI_MCC3_18C_ToPLC1 : E300ToMotor := (CommsOK := 1);
   AOI_MCC3_18E_ToPLC1 : E300ToMotor := (CommsOK := 1);
   AOI_MCC3_18G_ToPLC1 : E300ToMotor;
   AOI_MCC3_18J_ToPLC1 : E300ToMotor := (CommsOK := 1);
   AOI_MCC3_18L_ToPLC1 : E300ToMotor := (CommsOK := 1);
   AOI_MCC3_19A_ToPLC1 : E300ToMotor := (CommsOK := 1);
   AOI_MCC3_19C_ToPLC1 : E300ToMotor := (CommsOK := 1);
   AOI_MCC3_19E_ToPLC1 : E300ToMotor := (CommsOK := 1);
   AOI_MCC3_19G_ToPLC1 : E300ToMotor := (CommsOK := 1);
   AOI_MCC3_19J_ToPLC1 : E300ToMotor := (CommsOK := 1);
   AOI_MCC3_20A_ToPLC1 : E300ToMotor := (CommsOK := 1);
   AOI_MCC3_20C_ToPLC1 : E300ToMotor := (CommsOK := 1);
   AOI_MCC3_20E_ToPLC1 : E300ToMotor := (CommsOK := 1);
   AOI_MCC3_20G_ToPLC1 : E300ToMotor := (CommsOK := 1);
   AOI_MCC3_20J_ToPLC1 : E300ToMotor := (CommsOK := 1);
   AOI_MCC3_21A_ToPLC1 : E300ToMotor := (CommsOK := 1);
   AOI_MCC3_21C_ToPLC1 : E300ToMotor := (CommsOK := 1);
   AOI_MCC3_21E_ToPLC1 : E300ToMotor := (CommsOK := 1);
   AOI_MCC3_21G_ToPLC1 : E300ToMotor := (CommsOK := 1);
   AOI_MCC3_21J_ToPLC1 : E300ToMotor := (CommsOK := 1);
   AOI_MCC3_21L_ToPLC1 : E300ToMotor := (CommsOK := 1);
   AOI_MCC3_22C_ToPLC1 : E300ToMotor := (CommsOK := 1);
   AOI_MCC3_22E_ToPLC1 : E300ToMotor := (CommsOK := 1);
   AOI_MCC3_2A_ToPLC1 : PF525ToMotor := (CommsOK := 1);
   AOI_MCC3_2D_ToPLC1 : PF525ToMotor := (CommsOK := 1);
   AOI_MCC3_2G_ToPLC1 : PF525ToMotor := (CommsOK := 1);
   AOI_MCC3_2K_ToPLC1 : PF525ToMotor := (CommsOK := 1);
   AOI_MCC3_3A_ToPLC1 : PF525ToMotor := (CommsOK := 1);
   AOI_MCC3_3D_ToPLC1 : PF525ToMotor := (CommsOK := 1);
   AOI_MCC3_3G_ToPLC1 : PF525ToMotor := (CommsOK := 1);
   AOI_MCC3_3K_ToPLC1 : PF525ToMotor := (CommsOK := 1);
   AOI_MCC3_4A_ToPLC1 : PF525ToMotor := (CommsOK := 1);
   AOI_MCC3_4D_ToPLC1 : PF525ToMotor := (CommsOK := 1);
   AOI_MCC3_4G_ToPLC1 : PF525ToMotor := (CommsOK := 1);
   AOI_MCC3_4K_ToPLC1 : PF525ToMotor := (CommsOK := 1);
   AOI_MCC3_5A_ToPLC1 : PF525ToMotor := (CommsOK := 1);
   AOI_MCC3_5D_ToPLC1 : PF525ToMotor := (CommsOK := 1);
   AOI_MCC3_5G_ToPLC1 : PF525ToMotor := (CommsOK := 1);
   AOI_MCC3_5K_ToPLC1 : PF525ToMotor := (CommsOK := 1);
   AOI_MCC3_6A_ToPLC1 : PF525ToMotor := (CommsOK := 1);
   AOI_MCC3_6D_ToPLC1 : PF525ToMotor := (CommsOK := 1);
   AOI_MCC3_6G_ToPLC1 : E300ToMotor := (CommsOK := 1);
   AOI_MCC3_6J_ToPLC1 : E300ToMotor := (CommsOK := 1);
   AOI_MCC3_7A_ToPLC1 : E300ToMotor := (CommsOK := 1);
   AOI_MCC3_7C_ToPLC1 : E300ToMotor := (CommsOK := 1);
   AOI_MCC3_7E_ToPLC1 : E300ToMotor := (CommsOK := 1);
   AOI_MCC3_7G_ToPLC1 : PF525ToMotor := (CommsOK := 1);
   AOI_MCC3_7K_ToPLC1 : PF525ToMotor := (CommsOK := 1);
   AOI_MCC3_8A_ToPLC1 : E300ToMotor;
   AOI_MCC3_8D_ToPLC1 : PF525ToMotor := (CommsOK := 1);
   AOI_MCC3_8H_ToPLC1 : E300ToMotor;
   AOI_MCC3_8K_ToPLC1 : PF525ToMotor := (CommsOK := 1);
   AOI_MCC3_9A_ToPLC1 : E300ToMotor := (CommsOK := 1);
   AOI_MCC3_9C_ToPLC1 : E300ToMotor := (CommsOK := 1);
   AOI_MCC3_9E_ToPLC1 : E300ToMotor := (CommsOK := 1);
   AOI_MCC3_9G_ToPLC1 : E300ToMotor := (CommsOK := 1);
   AOI_MCC3_9J_ToPLC1 : E300ToMotor := (CommsOK := 1);
   AOI_MCC3_9L_ToPLC1 : E300ToMotor;
   AOI_MCC4_1E_ToPLC1 : PF525ToMotor := (CommsOK := 1);
   AOI_MCC4_2A_ToPLC1 : E300ToMotor := (CommsOK := 1);
   AOI_MCC4_2C_ToPLC1 : E300ToMotor := (CommsOK := 1);
   AOI_MCC4_2E_ToPLC1 : E300ToMotor := (CommsOK := 1);
   AOI_MCC4_2G_ToPLC1 : PF525ToMotor;
   AOI_MCC4_2K_ToPLC1 : PF525ToMotor := (CommsOK := 1);
   AOI_MCC4_3A_ToPLC1 : E300ToMotor := (CommsOK := 1);
   AOI_MCC4_3C_ToPLC1 : E300ToMotor := (CommsOK := 1);
   AOI_MCC4_3E_ToPLC1 : E300ToMotor := (CommsOK := 1);
   AOI_MCC4_3G_ToPLC1 : E300ToMotor := (CommsOK := 1);
   AOI_MCC4_3J_ToPLC1 : E300ToMotor := (CommsOK := 1);
   AOI_MCC4_3L_ToPLC1 : E300ToMotor := (CommsOK := 1);
   AOI_MCC4_4A_ToPLC1 : E300ToMotor;
   AOI_MCC4_4C_ToPLC1 : E300ToMotor := (CommsOK := 1);
   AOI_MCC4_4E_ToPLC1 : E300ToMotor;
   AOI_MCC4_4G_ToPLC1 : E300ToMotor;
   AOI_MCC4_4J_ToPLC1 : E300ToMotor;
   AOI_MCC4_4L_ToPLC1 : E300ToMotor;
   AOI_MCC4_5A_ToPLC1 : E300ToMotor;
   AOI_MCC4_5C_ToPLC1 : E300ToMotor := (CommsOK := 1);
   AOI_MCC4_5E_ToPLC1 : E300ToMotor;
   AOI_PLC1_To_MCC2_10A : MotorToE300 := (OK := 1);
   AOI_PLC1_To_MCC2_10C : MotorToE300 := (OK := 1);
   AOI_PLC1_To_MCC2_10E : MotorToE300 := (OK := 1);
   AOI_PLC1_To_MCC2_10G : MotorToE300 := (OK := 1);
   AOI_PLC1_To_MCC2_10J : MotorToE300 := (OK := 1);
   AOI_PLC1_To_MCC2_10L : MotorToE300 := (OK := 1);
   AOI_PLC1_To_MCC2_11A : MotorToE300 := (OK := 1);
   AOI_PLC1_To_MCC2_11C : MotorToE300 := (OK := 1);
   AOI_PLC1_To_MCC2_11E : MotorToE300 := (OK := 1);
   AOI_PLC1_To_MCC2_11G : MotorToE300 := (OK := 1);
   AOI_PLC1_To_MCC2_11J : MotorToE300 := (OK := 1);
   AOI_PLC1_To_MCC2_11L : MotorToE300 := (OK := 1);
   AOI_PLC1_To_MCC2_12A : MotorToE300 := (OK := 1);
   AOI_PLC1_To_MCC2_12C : MotorToE300 := (OK := 1);
   AOI_PLC1_To_MCC2_12E : MotorToE300 := (OK := 1);
   AOI_PLC1_To_MCC2_12G : MotorToE300 := (OK := 1);
   AOI_PLC1_To_MCC2_12J : MotorToE300 := (OK := 1);
   AOI_PLC1_To_MCC2_12L : MotorToE300 := (OK := 1);
   AOI_PLC1_To_MCC2_13A : MotorToE300 := (OK := 1);
   AOI_PLC1_To_MCC2_13C : MotorToE300 := (OK := 1);
   AOI_PLC1_To_MCC2_13E : MotorToE300 := (OK := 1);
   AOI_PLC1_To_MCC2_13G : MotorToE300 := (OK := 1);
   AOI_PLC1_To_MCC2_13J : MotorToE300 := (OK := 1);
   AOI_PLC1_To_MCC2_14A : MotorToE300 := (OK := 1);
   AOI_PLC1_To_MCC2_14C : MotorToE300 := (OK := 1);
   AOI_PLC1_To_MCC2_14E : MotorToE300 := (OK := 1);
   AOI_PLC1_To_MCC2_14G : MotorToE300 := (OK := 1);
   AOI_PLC1_To_MCC2_14J : MotorToE300 := (OK := 1);
   AOI_PLC1_To_MCC2_14L : MotorToE300 := (OK := 1);
   AOI_PLC1_To_MCC2_15A : MotorToE300 := (OK := 1);
   AOI_PLC1_To_MCC2_15C : MotorToE300 := (OK := 1);
   AOI_PLC1_To_MCC2_15E : MotorToE300 := (OK := 1);
   AOI_PLC1_To_MCC2_15G : MotorToE300 := (OK := 1);
   AOI_PLC1_To_MCC2_15J : MotorToE300 := (OK := 1);
   AOI_PLC1_To_MCC2_15L : MotorToE300 := (OK := 1);
   AOI_PLC1_To_MCC2_16A : MotorToE300 := (OK := 1);
   AOI_PLC1_To_MCC2_16C : MotorToE300 := (OK := 1);
   AOI_PLC1_To_MCC2_16E : MotorToE300 := (OK := 1);
   AOI_PLC1_To_MCC2_16G : MotorToE300 := (OK := 1);
   AOI_PLC1_To_MCC2_16J : MotorToE300 := (OK := 1);
   AOI_PLC1_To_MCC2_16L : MotorToE300 := (OK := 1);
   AOI_PLC1_To_MCC2_17A : MotorToE300 := (OK := 1);
   AOI_PLC1_To_MCC2_17C : MotorToE300 := (OK := 1);
   AOI_PLC1_To_MCC2_17E : MotorToE300 := (OK := 1);
   AOI_PLC1_To_MCC2_17G : MotorToE300 := (OK := 1);
   AOI_PLC1_To_MCC2_17J : MotorToE300 := (OK := 1);
   AOI_PLC1_To_MCC2_18A : MotorToE300 := (OK := 1);
   AOI_PLC1_To_MCC2_18C : MotorToE300 := (OK := 1);
   AOI_PLC1_To_MCC2_18E : MotorToE300 := (OK := 1);
   AOI_PLC1_To_MCC2_18G : MotorToE300 := (OK := 1);
   AOI_PLC1_To_MCC2_18J : MotorToE300 := (OK := 1);
   AOI_PLC1_To_MCC2_18L : MotorToE300 := (OK := 1);
   AOI_PLC1_To_MCC2_19A : MotorToE300 := (OK := 1);
   AOI_PLC1_To_MCC2_19C : MotorToE300 := (OK := 1);
   AOI_PLC1_To_MCC2_19E : MotorToE300 := (OK := 1);
   AOI_PLC1_To_MCC2_19G : MotorToE300 := (OK := 1);
   AOI_PLC1_To_MCC2_19J : MotorToE300 := (OK := 1);
   AOI_PLC1_To_MCC2_19L : MotorToE300 := (OK := 1);
   AOI_PLC1_To_MCC2_20C : MotorToE300 := (OK := 1);
   AOI_PLC1_To_MCC2_20E : MotorToE300 := (OK := 1);
   AOI_PLC1_To_MCC2_20G : MotorToE300 := (OK := 1);
   AOI_PLC1_To_MCC2_20J : MotorToE300 := (OK := 1);
   AOI_PLC1_To_MCC2_21A : MotorToE300 := (OK := 1);
   AOI_PLC1_To_MCC2_21C : MotorToE300 := (OK := 1);
   AOI_PLC1_To_MCC2_21E : MotorToE300 := (OK := 1);
   AOI_PLC1_To_MCC2_21G : MotorToPF525 := (OK := 1);
   AOI_PLC1_To_MCC2_21K : MotorToPF525 := (OK := 1);
   AOI_PLC1_To_MCC2_2A : MotorToPF525 := (OK := 1);   // Motor From PLC1 to PF525 AOI
   AOI_PLC1_To_MCC2_2D : MotorToPF525 := (OK := 1);
   AOI_PLC1_To_MCC2_2G : MotorToPF525 := (OK := 1);
   AOI_PLC1_To_MCC2_2K : MotorToPF525 := (OK := 1);
   AOI_PLC1_To_MCC2_3A : MotorToE300 := (OK := 1);
   AOI_PLC1_To_MCC2_3C : MotorToE300 := (OK := 1);
   AOI_PLC1_To_MCC2_3E : MotorToE300 := (OK := 1);
   AOI_PLC1_To_MCC2_3G : MotorToE300 := (OK := 1);
   AOI_PLC1_To_MCC2_3J : MotorToE300 := (OK := 1);
   AOI_PLC1_To_MCC2_3L : MotorToE300 := (OK := 1);
   AOI_PLC1_To_MCC2_4A : MotorToE300 := (OK := 1);
   AOI_PLC1_To_MCC2_4C : MotorToE300 := (OK := 1);
   AOI_PLC1_To_MCC2_4E : MotorToE300 := (OK := 1);
   AOI_PLC1_To_MCC2_4G : MotorToE300 := (OK := 1);
   AOI_PLC1_To_MCC2_4J : MotorToE300 := (OK := 1);
   AOI_PLC1_To_MCC2_4L : MotorToE300 := (OK := 1);
   AOI_PLC1_To_MCC2_5A : MotorToE300 := (OK := 1);
   AOI_PLC1_To_MCC2_5C : MotorToE300 := (OK := 1);
   AOI_PLC1_To_MCC2_5E : MotorToE300 := (OK := 1);
   AOI_PLC1_To_MCC2_5G : MotorToE300 := (OK := 1);
   AOI_PLC1_To_MCC2_5J : MotorToE300 := (OK := 1);
   AOI_PLC1_To_MCC2_6A : MotorToE300 := (OK := 1);
   AOI_PLC1_To_MCC2_6C : MotorToE300 := (OK := 1);
   AOI_PLC1_To_MCC2_6E : MotorToE300 := (OK := 1);
   AOI_PLC1_To_MCC2_6G : MotorToE300 := (OK := 1);
   AOI_PLC1_To_MCC2_6J : MotorToE300 := (OK := 1);
   AOI_PLC1_To_MCC2_6L : MotorToE300 := (OK := 1);
   AOI_PLC1_To_MCC2_7A : MotorToE300 := (OK := 1);
   AOI_PLC1_To_MCC2_7D : MotorToE300 := (OK := 1);
   AOI_PLC1_To_MCC2_7G : MotorToE300 := (OK := 1);
   AOI_PLC1_To_MCC2_7K : MotorToE300 := (OK := 1);
   AOI_PLC1_To_MCC2_8B : MotorToE300 := (OK := 1);
   AOI_PLC1_To_MCC2_8D : MotorToE300 := (OK := 1);
   AOI_PLC1_To_MCC2_8F : MotorToE300 := (OK := 1);
   AOI_PLC1_To_MCC2_8H : MotorToE300 := (OK := 1);
   AOI_PLC1_To_MCC2_8K : MotorToE300 := (OK := 1);
   AOI_PLC1_To_MCC2_9D : MotorToE300 := (OK := 1);
   AOI_PLC1_To_MCC2_9F : MotorToE300 := (OK := 1);
   AOI_PLC1_To_MCC2_9H : MotorToPF525 := (OK := 1);
   AOI_PLC1_To_MCC3_10A : MotorToE300 := (OK := 1);
   AOI_PLC1_To_MCC3_10D : MotorToE300 := (OK := 1);
   AOI_PLC1_To_MCC3_10G : MotorToE300 := (OK := 1);
   AOI_PLC1_To_MCC3_10J : MotorToE300 := (OK := 1);
   AOI_PLC1_To_MCC3_11A : MotorToE300 := (OK := 1);
   AOI_PLC1_To_MCC3_11D : MotorToE300 := (OK := 1);
   AOI_PLC1_To_MCC3_11G : MotorToE300 := (OK := 1);
   AOI_PLC1_To_MCC3_11J : MotorToE300 := (OK := 1);
   AOI_PLC1_To_MCC3_12A : MotorToE300 := (OK := 1);
   AOI_PLC1_To_MCC3_12C : MotorToE300 := (OK := 1);
   AOI_PLC1_To_MCC3_12E : MotorToE300 := (OK := 1);
   AOI_PLC1_To_MCC3_12G : MotorToE300 := (OK := 1);
   AOI_PLC1_To_MCC3_12J : MotorToE300 := (OK := 1);
   AOI_PLC1_To_MCC3_12L : MotorToE300 := (OK := 1);
   AOI_PLC1_To_MCC3_13A : MotorToE300 := (OK := 1);
   AOI_PLC1_To_MCC3_13C : MotorToE300 := (OK := 1);
   AOI_PLC1_To_MCC3_13E : MotorToE300 := (OK := 1);
   AOI_PLC1_To_MCC3_13G : MotorToE300 := (OK := 1);
   AOI_PLC1_To_MCC3_13J : MotorToE300 := (OK := 1);
   AOI_PLC1_To_MCC3_13L : MotorToE300 := (OK := 1);
   AOI_PLC1_To_MCC3_14A : MotorToE300 := (OK := 1);
   AOI_PLC1_To_MCC3_14C : MotorToE300 := (OK := 1);
   AOI_PLC1_To_MCC3_14E : MotorToE300 := (OK := 1);
   AOI_PLC1_To_MCC3_14G : MotorToE300 := (OK := 1);
   AOI_PLC1_To_MCC3_14J : MotorToE300 := (OK := 1);
   AOI_PLC1_To_MCC3_14L : MotorToE300 := (OK := 1);
   AOI_PLC1_To_MCC3_15A : MotorToE300 := (OK := 1);
   AOI_PLC1_To_MCC3_15C : MotorToE300 := (OK := 1);
   AOI_PLC1_To_MCC3_15E : MotorToE300 := (OK := 1);
   AOI_PLC1_To_MCC3_15G : MotorToE300 := (OK := 1);
   AOI_PLC1_To_MCC3_15J : MotorToE300 := (OK := 1);
   AOI_PLC1_To_MCC3_16A : MotorToE300 := (OK := 1);
   AOI_PLC1_To_MCC3_16C : MotorToE300 := (OK := 1);
   AOI_PLC1_To_MCC3_16E : MotorToE300 := (OK := 1);
   AOI_PLC1_To_MCC3_16G : MotorToE300 := (OK := 1);
   AOI_PLC1_To_MCC3_16J : MotorToE300 := (OK := 1);
   AOI_PLC1_To_MCC3_16L : MotorToE300 := (OK := 1);
   AOI_PLC1_To_MCC3_17A : MotorToE300 := (OK := 1);
   AOI_PLC1_To_MCC3_17C : MotorToE300 := (OK := 1);
   AOI_PLC1_To_MCC3_17E : MotorToE300 := (OK := 1);
   AOI_PLC1_To_MCC3_17G : MotorToE300 := (OK := 1);
   AOI_PLC1_To_MCC3_17J : MotorToE300 := (OK := 1);
   AOI_PLC1_To_MCC3_17L : MotorToE300 := (OK := 1);
   AOI_PLC1_To_MCC3_18A : MotorToE300 := (OK := 1);
   AOI_PLC1_To_MCC3_18C : MotorToE300 := (OK := 1);
   AOI_PLC1_To_MCC3_18E : MotorToE300 := (OK := 1);
   AOI_PLC1_To_MCC3_18G : MotorToE300 := (OK := 1);
   AOI_PLC1_To_MCC3_18J : MotorToE300 := (OK := 1);
   AOI_PLC1_To_MCC3_18L : MotorToE300 := (OK := 1);
   AOI_PLC1_To_MCC3_19A : MotorToE300 := (OK := 1);
   AOI_PLC1_To_MCC3_19C : MotorToE300 := (OK := 1);
   AOI_PLC1_To_MCC3_19E : MotorToE300 := (OK := 1);
   AOI_PLC1_To_MCC3_19G : MotorToE300 := (OK := 1);
   AOI_PLC1_To_MCC3_19J : MotorToE300 := (OK := 1);
   AOI_PLC1_To_MCC3_20A : MotorToE300 := (OK := 1);
   AOI_PLC1_To_MCC3_20C : MotorToE300 := (OK := 1);
   AOI_PLC1_To_MCC3_20E : MotorToE300 := (OK := 1);
   AOI_PLC1_To_MCC3_20G : MotorToE300 := (OK := 1);
   AOI_PLC1_To_MCC3_20J : MotorToE300 := (OK := 1);
   AOI_PLC1_To_MCC3_21A : MotorToE300 := (OK := 1);
   AOI_PLC1_To_MCC3_21C : MotorToE300 := (OK := 1);
   AOI_PLC1_To_MCC3_21E : MotorToE300 := (OK := 1);
   AOI_PLC1_To_MCC3_21G : MotorToE300 := (OK := 1);
   AOI_PLC1_To_MCC3_21J : MotorToE300 := (OK := 1);
   AOI_PLC1_To_MCC3_21L : MotorToE300 := (OK := 1);
   AOI_PLC1_To_MCC3_22C : MotorToE300 := (OK := 1);
   AOI_PLC1_To_MCC3_22E : MotorToE300 := (OK := 1);
   AOI_PLC1_To_MCC3_2A : MotorToPF525 := (OK := 1);
   AOI_PLC1_To_MCC3_2D : MotorToPF525 := (OK := 1);
   AOI_PLC1_To_MCC3_2G : MotorToPF525 := (OK := 1);
   AOI_PLC1_To_MCC3_2K : MotorToPF525 := (OK := 1);
   AOI_PLC1_To_MCC3_3A : MotorToPF525 := (OK := 1);
   AOI_PLC1_To_MCC3_3D : MotorToPF525 := (OK := 1);
   AOI_PLC1_To_MCC3_3G : MotorToPF525 := (OK := 1);
   AOI_PLC1_To_MCC3_3K : MotorToPF525 := (OK := 1);
   AOI_PLC1_To_MCC3_4A : MotorToPF525 := (OK := 1);
   AOI_PLC1_To_MCC3_4D : MotorToPF525 := (OK := 1);
   AOI_PLC1_To_MCC3_4G : MotorToPF525 := (OK := 1);
   AOI_PLC1_To_MCC3_4K : MotorToPF525 := (OK := 1);
   AOI_PLC1_To_MCC3_5A : MotorToPF525 := (OK := 1);
   AOI_PLC1_To_MCC3_5D : MotorToPF525 := (OK := 1);
   AOI_PLC1_To_MCC3_5G : MotorToPF525 := (OK := 1);
   AOI_PLC1_To_MCC3_5K : MotorToPF525 := (OK := 1);
   AOI_PLC1_To_MCC3_6A : MotorToPF525 := (OK := 1);
   AOI_PLC1_To_MCC3_6D : MotorToPF525 := (OK := 1);
   AOI_PLC1_To_MCC3_6G : MotorToE300 := (OK := 1);
   AOI_PLC1_To_MCC3_6J : MotorToE300 := (OK := 1);
   AOI_PLC1_To_MCC3_7A : MotorToE300 := (OK := 1);
   AOI_PLC1_To_MCC3_7C : MotorToE300 := (OK := 1);
   AOI_PLC1_To_MCC3_7E : MotorToE300 := (OK := 1);
   AOI_PLC1_To_MCC3_7G : MotorToPF525 := (OK := 1);
   AOI_PLC1_To_MCC3_7K : MotorToPF525 := (OK := 1);
   AOI_PLC1_To_MCC3_8A : MotorToE300 := (OK := 1);
   AOI_PLC1_To_MCC3_8D : MotorToPF525 := (OK := 1);
   AOI_PLC1_To_MCC3_8H : MotorToE300 := (OK := 1);
   AOI_PLC1_To_MCC3_8K : MotorToPF525 := (OK := 1);
   AOI_PLC1_To_MCC3_9A : MotorToE300 := (OK := 1);
   AOI_PLC1_To_MCC3_9C : MotorToE300 := (OK := 1);
   AOI_PLC1_To_MCC3_9E : MotorToE300 := (OK := 1);
   AOI_PLC1_To_MCC3_9G : MotorToE300 := (OK := 1);
   AOI_PLC1_To_MCC3_9J : MotorToE300 := (OK := 1);
   AOI_PLC1_To_MCC3_9L : MotorToE300 := (OK := 1);
   AOI_PLC1_To_MCC4_1E : MotorToPF525 := (OK := 1);
   AOI_PLC1_To_MCC4_2A : MotorToE300 := (OK := 1);
   AOI_PLC1_To_MCC4_2C : MotorToE300 := (OK := 1);
   AOI_PLC1_To_MCC4_2E : MotorToE300 := (OK := 1);
   AOI_PLC1_To_MCC4_2G : MotorToPF525 := (OK := 1);
   AOI_PLC1_To_MCC4_2K : MotorToPF525 := (OK := 1);
   AOI_PLC1_To_MCC4_3A : MotorToE300 := (OK := 1);
   AOI_PLC1_To_MCC4_3C : MotorToE300 := (OK := 1);
   AOI_PLC1_To_MCC4_3E : MotorToE300 := (OK := 1);
   AOI_PLC1_To_MCC4_3G : MotorToE300 := (OK := 1);
   AOI_PLC1_To_MCC4_3J : MotorToE300 := (OK := 1);
   AOI_PLC1_To_MCC4_3L : MotorToE300 := (OK := 1);
   AOI_PLC1_To_MCC4_4A : MotorToE300 := (OK := 1);
   AOI_PLC1_To_MCC4_4C : MotorToE300 := (OK := 1);
   AOI_PLC1_To_MCC4_4E : MotorToE300 := (OK := 1);
   AOI_PLC1_To_MCC4_4G : MotorToE300 := (OK := 1);
   AOI_PLC1_To_MCC4_4J : MotorToE300 := (OK := 1);
   AOI_PLC1_To_MCC4_4L : MotorToE300 := (OK := 1);
   AOI_PLC1_To_MCC4_5A : MotorToE300 := (OK := 1);
   AOI_PLC1_To_MCC4_5C : MotorToE300 := (OK := 1);
   AOI_PLC1_To_MCC4_5E : MotorToE300 := (OK := 1);
   Const_4000_Hex : INT := 16384;   // Constant #16:4000, Entry Status Communicating
   GSV_EntryStatus : INT := 16384;   // GSV Entry Status, shold be #16:4000
   MCC2_10A_CommsOK : BOOL := 1;   // Communications with AOP OK
   MCC2_10C_CommsOK : BOOL := 1;   // Communications with AOP OK
   MCC2_10E_CommsOK : BOOL := 1;   // Communications with AOP OK
   MCC2_10G_CommsOK : BOOL := 1;   // Communications with AOP OK
   MCC2_10J_CommsOK : BOOL := 1;   // Communications with AOP OK
   MCC2_10L_CommsOK : BOOL := 1;   // Communications with AOP OK
   MCC2_11A_CommsOK : BOOL := 1;   // Communications with AOP OK
   MCC2_11C_CommsOK : BOOL := 1;   // Communications with AOP OK
   MCC2_11E_CommsOK : BOOL := 1;   // Communications with AOP OK
   MCC2_11G_CommsOK : BOOL := 1;   // Communications with AOP OK
   MCC2_11J_CommsOK : BOOL := 1;   // Communications with AOP OK
   MCC2_11L_CommsOK : BOOL;   // Communications with AOP OK
   MCC2_12A_CommsOK : BOOL := 1;   // Communications with AOP OK
   MCC2_12C_CommsOK : BOOL := 1;   // Communications with AOP OK
   MCC2_12E_CommsOK : BOOL := 1;   // Communications with AOP OK
   MCC2_12G_CommsOK : BOOL := 1;   // Communications with AOP OK
   MCC2_12J_CommsOK : BOOL := 1;   // Communications with AOP OK
   MCC2_12L_CommsOK : BOOL := 1;   // Communications with AOP OK
   MCC2_13A_CommsOK : BOOL := 1;   // Communications with AOP OK
   MCC2_13C_CommsOK : BOOL := 1;   // Communications with AOP OK
   MCC2_13E_CommsOK : BOOL;   // Communications with AOP OK
   MCC2_13G_CommsOK : BOOL := 1;   // Communications with AOP OK
   MCC2_13J_CommsOK : BOOL := 1;   // Communications with AOP OK
   MCC2_14A_CommsOK : BOOL := 1;   // Communications with AOP OK
   MCC2_14C_CommsOK : BOOL := 1;   // Communications with AOP OK
   MCC2_14E_CommsOK : BOOL := 1;   // Communications with AOP OK
   MCC2_14G_CommsOK : BOOL := 1;   // Communications with AOP OK
   MCC2_14J_CommsOK : BOOL;   // Communications with AOP OK
   MCC2_14L_CommsOK : BOOL := 1;   // Communications with AOP OK
   MCC2_15A_CommsOK : BOOL := 1;   // Communications with AOP OK
   MCC2_15C_CommsOK : BOOL := 1;   // Communications with AOP OK
   MCC2_15E_CommsOK : BOOL := 1;   // Communications with AOP OK
   MCC2_15G_CommsOK : BOOL := 1;   // Communications with AOP OK
   MCC2_15J_CommsOK : BOOL := 1;   // Communications with AOP OK
   MCC2_15L_CommsOK : BOOL := 1;   // Communications with AOP OK
   MCC2_16A_CommsOK : BOOL := 1;   // Communications with AOP OK
   MCC2_16C_CommsOK : BOOL := 1;   // Communications with AOP OK
   MCC2_16E_CommsOK : BOOL := 1;   // Communications with AOP OK
   MCC2_16G_CommsOK : BOOL := 1;   // Communications with AOP OK
   MCC2_16J_CommsOK : BOOL := 1;   // Communications with AOP OK
   MCC2_16L_CommsOK : BOOL := 1;   // Communications with AOP OK
   MCC2_17A_CommsOK : BOOL := 1;   // Communications with AOP OK
   MCC2_17C_CommsOK : BOOL := 1;   // Communications with AOP OK
   MCC2_17E_CommsOK : BOOL := 1;   // Communications with AOP OK
   MCC2_17G_CommsOK : BOOL := 1;   // Communications with AOP OK
   MCC2_17J_CommsOK : BOOL := 1;   // Communications with AOP OK
   MCC2_18A_CommsOK : BOOL := 1;   // Communications with AOP OK
   MCC2_18C_CommsOK : BOOL := 1;   // Communications with AOP OK
   MCC2_18E_CommsOK : BOOL := 1;   // Communications with AOP OK
   MCC2_18G_CommsOK : BOOL := 1;   // Communications with AOP OK
   MCC2_18J_CommsOK : BOOL := 1;   // Communications with AOP OK
   MCC2_18L_CommsOK : BOOL := 1;   // Communications with AOP OK
   MCC2_19A_CommsOK : BOOL := 1;   // Communications with AOP OK
   MCC2_19C_CommsOK : BOOL := 1;   // Communications with AOP OK
   MCC2_19E_CommsOK : BOOL := 1;   // Communications with AOP OK
   MCC2_19G_CommsOK : BOOL := 1;   // Communications with AOP OK
   MCC2_19J_CommsOK : BOOL := 1;   // Communications with AOP OK
   MCC2_19L_CommsOK : BOOL := 1;   // Communications with AOP OK
   MCC2_20C_CommsOK : BOOL := 1;   // Communications with AOP OK
   MCC2_20E_CommsOK : BOOL := 1;   // Communications with AOP OK
   MCC2_20G_CommsOK : BOOL;   // Communications with AOP OK
   MCC2_20J_CommsOK : BOOL := 1;   // Communications with AOP OK
   MCC2_21A_CommsOK : BOOL := 1;   // Communications with AOP OK
   MCC2_21C_CommsOK : BOOL := 1;   // Communications with AOP OK
   MCC2_21E_CommsOK : BOOL := 1;   // Communications with AOP OK
   MCC2_21G_CommsOK : BOOL := 1;   // Communications with AOP OK
   MCC2_21K_CommsOK : BOOL;   // Communications with AOP OK
   MCC2_2A_CommsOK : BOOL := 1;   // Communications with AOP OK
   MCC2_2D_CommsOK : BOOL := 1;   // Communications with AOP OK
   MCC2_2G_CommsOK : BOOL := 1;   // Communications with AOP OK
   MCC2_2K_CommsOK : BOOL := 1;   // Communications with AOP OK
   MCC2_3A_CommsOK : BOOL := 1;   // Communications with AOP OK
   MCC2_3C_CommsOK : BOOL := 1;   // Communications with AOP OK
   MCC2_3E_CommsOK : BOOL := 1;   // Communications with AOP OK
   MCC2_3G_CommsOK : BOOL := 1;   // Communications with AOP OK
   MCC2_3J_CommsOK : BOOL := 1;   // Communications with AOP OK
   MCC2_3L_CommsOK : BOOL := 1;   // Communications with AOP OK
   MCC2_4A_CommsOK : BOOL := 1;   // Communications with AOP OK
   MCC2_4C_CommsOK : BOOL := 1;   // Communications with AOP OK
   MCC2_4E_CommsOK : BOOL := 1;   // Communications with AOP OK
   MCC2_4G_CommsOK : BOOL := 1;   // Communications with AOP OK
   MCC2_4J_CommsOK : BOOL := 1;   // Communications with AOP OK
   MCC2_4L_CommsOK : BOOL := 1;   // Communications with AOP OK
   MCC2_5A_CommsOK : BOOL := 1;   // Communications with AOP OK
   MCC2_5C_CommsOK : BOOL := 1;   // Communications with AOP OK
   MCC2_5E_CommsOK : BOOL := 1;   // Communications with AOP OK
   MCC2_5G_CommsOK : BOOL := 1;   // Communications with AOP OK
   MCC2_5J_CommsOK : BOOL := 1;   // Communications with AOP OK
   MCC2_6A_CommsOK : BOOL := 1;   // Communications with AOP OK
   MCC2_6C_CommsOK : BOOL := 1;   // Communications with AOP OK
   MCC2_6E_CommsOK : BOOL := 1;   // Communications with AOP OK
   MCC2_6G_CommsOK : BOOL := 1;   // Communications with AOP OK
   MCC2_6J_CommsOK : BOOL := 1;   // Communications with AOP OK
   MCC2_6L_CommsOK1 : BOOL := 1;   // Communications with AOP OK
   MCC2_7A_CommsOK : BOOL := 1;   // Communications with AOP OK
   MCC2_7D_CommsOK : BOOL := 1;   // Communications with AOP OK
   MCC2_7G_CommsOK : BOOL := 1;   // Communications with AOP OK
   MCC2_7K_CommsOK : BOOL;   // Communications with AOP OK
   MCC2_8B_CommsOK : BOOL;   // Communications with AOP OK
   MCC2_8D_CommsOK : BOOL := 1;   // Communications with AOP OK
   MCC2_8F_CommsOK : BOOL := 1;   // Communications with AOP OK
   MCC2_8H_CommsOK : BOOL := 1;   // Communications with AOP OK
   MCC2_8K_CommsOK : BOOL;   // Communications with AOP OK
   MCC2_9D_CommsOK : BOOL := 1;   // Communications with AOP OK
   MCC2_9F_CommsOK : BOOL := 1;   // Communications with AOP OK
   MCC2_9H_CommsOK : BOOL := 1;   // Communications with AOP OK
   MCC3_10A_CommsOK : BOOL := 1;   // Communications with AOP OK
   MCC3_10D_CommsOK : BOOL;   // Communications with AOP OK
   MCC3_10G_CommsOK : BOOL := 1;   // Communications with AOP OK
   MCC3_10J_CommsOK : BOOL;   // Communications with AOP OK
   MCC3_11A_CommsOK : BOOL := 1;   // Communications with AOP OK
   MCC3_11D_CommsOK : BOOL := 1;   // Communications with AOP OK
   MCC3_11G_CommsOK : BOOL := 1;   // Communications with AOP OK
   MCC3_11J_CommsOK : BOOL;   // Communications with AOP OK
   MCC3_12A_CommsOK : BOOL;   // Communications with AOP OK
   MCC3_12C_CommsOK : BOOL := 1;   // Communications with AOP OK
   MCC3_12E_CommsOK : BOOL := 1;   // Communications with AOP OK
   MCC3_12G_CommsOK : BOOL := 1;   // Communications with AOP OK
   MCC3_12J_CommsOK : BOOL := 1;   // Communications with AOP OK
   MCC3_12L_CommsOK : BOOL := 1;   // Communications with AOP OK
   MCC3_13A_CommsOK : BOOL := 1;   // Communications with AOP OK
   MCC3_13C_CommsOK : BOOL := 1;   // Communications with AOP OK
   MCC3_13E_CommsOK : BOOL := 1;   // Communications with AOP OK
   MCC3_13G_CommsOK : BOOL := 1;   // Communications with AOP OK
   MCC3_13J_CommsOK : BOOL := 1;   // Communications with AOP OK
   MCC3_13L_CommsOK : BOOL := 1;   // Communications with AOP OK
   MCC3_14A_CommsOK : BOOL := 1;   // Communications with AOP OK
   MCC3_14C_CommsOK : BOOL := 1;   // Communications with AOP OK
   MCC3_14E_CommsOK : BOOL := 1;   // Communications with AOP OK
   MCC3_14G_CommsOK : BOOL := 1;   // Communications with AOP OK
   MCC3_14J_CommsOK : BOOL := 1;   // Communications with AOP OK
   MCC3_14L_CommsOK : BOOL;   // Communications with AOP OK
   MCC3_15A_CommsOK : BOOL := 1;   // Communications with AOP OK
   MCC3_15C_CommsOK : BOOL := 1;   // Communications with AOP OK
   MCC3_15E_CommsOK : BOOL := 1;   // Communications with AOP OK
   MCC3_15G_CommsOK : BOOL := 1;   // Communications with AOP OK
   MCC3_15J_CommsOK : BOOL;   // Communications with AOP OK
   MCC3_16A_CommsOK : BOOL := 1;   // Communications with AOP OK
   MCC3_16C_CommsOK : BOOL := 1;   // Communications with AOP OK
   MCC3_16E_CommsOK : BOOL;   // Communications with AOP OK
   MCC3_16G_CommsOK : BOOL := 1;   // Communications with AOP OK
   MCC3_16J_CommsOK : BOOL := 1;   // Communications with AOP OK
   MCC3_16L_CommsOK : BOOL := 1;   // Communications with AOP OK
   MCC3_17A_CommsOK : BOOL := 1;   // Communications with AOP OK
   MCC3_17C_CommsOK : BOOL := 1;   // Communications with AOP OK
   MCC3_17E_CommsOK : BOOL := 1;   // Communications with AOP OK
   MCC3_17G_CommsOK : BOOL := 1;   // Communications with AOP OK
   MCC3_17J_CommsOK : BOOL := 1;   // Communications with AOP OK
   MCC3_17L_CommsOK : BOOL := 1;   // Communications with AOP OK
   MCC3_18A_CommsOK : BOOL := 1;   // Communications with AOP OK
   MCC3_18C_CommsOK : BOOL := 1;   // Communications with AOP OK
   MCC3_18E_CommsOK : BOOL := 1;   // Communications with AOP OK
   MCC3_18G_CommsOK : BOOL;   // Communications with AOP OK
   MCC3_18J_CommsOK : BOOL := 1;   // Communications with AOP OK
   MCC3_18L_CommsOK : BOOL := 1;   // Communications with AOP OK
   MCC3_19A_CommsOK : BOOL := 1;   // Communications with AOP OK
   MCC3_19C_CommsOK : BOOL := 1;   // Communications with AOP OK
   MCC3_19E_CommsOK : BOOL := 1;   // Communications with AOP OK
   MCC3_19G_CommsOK : BOOL := 1;   // Communications with AOP OK
   MCC3_19J_CommsOK : BOOL := 1;   // Communications with AOP OK
   MCC3_20A_CommsOK : BOOL := 1;   // Communications with AOP OK
   MCC3_20C_CommsOK : BOOL := 1;   // Communications with AOP OK
   MCC3_20E_CommsOK : BOOL := 1;   // Communications with AOP OK
   MCC3_20G_CommsOK : BOOL := 1;   // Communications with AOP OK
   MCC3_20J_CommsOK : BOOL := 1;   // Communications with AOP OK
   MCC3_21A_CommsOK : BOOL := 1;   // Communications with AOP OK
   MCC3_21C_CommsOK : BOOL := 1;   // Communications with AOP OK
   MCC3_21E_CommsOK : BOOL := 1;   // Communications with AOP OK
   MCC3_21G_CommsOK : BOOL := 1;   // Communications with AOP OK
   MCC3_21J_CommsOK : BOOL := 1;   // Communications with AOP OK
   MCC3_21L_CommsOK : BOOL := 1;   // Communications with AOP OK
   MCC3_22C_CommsOK : BOOL := 1;   // Communications with AOP OK
   MCC3_22E_CommsOK : BOOL := 1;   // Communications with AOP OK
   MCC3_2A_CommsOK : BOOL := 1;   // Communications with AOP OK
   MCC3_2D_CommsOK : BOOL := 1;   // Communications with AOP OK
   MCC3_2G_CommsOK : BOOL := 1;   // Communications with AOP OK
   MCC3_2K_CommsOK : BOOL := 1;   // Communications with AOP OK
   MCC3_3A_CommsOK : BOOL := 1;   // Communications with AOP OK
   MCC3_3D_CommsOK : BOOL := 1;   // Communications with AOP OK
   MCC3_3G_CommsOK : BOOL := 1;   // Communications with AOP OK
   MCC3_3K_CommsOK : BOOL := 1;   // Communications with AOP OK
   MCC3_4A_CommsOK : BOOL := 1;   // Communications with AOP OK
   MCC3_4D_CommsOK : BOOL := 1;   // Communications with AOP OK
   MCC3_4G_CommsOK : BOOL := 1;   // Communications with AOP OK
   MCC3_4K_CommsOK : BOOL := 1;   // Communications with AOP OK
   MCC3_5A_CommsOK : BOOL := 1;   // Communications with AOP OK
   MCC3_5D_CommsOK : BOOL := 1;   // Communications with AOP OK
   MCC3_5G_CommsOK : BOOL := 1;   // Communications with AOP OK
   MCC3_5K_CommsOK : BOOL := 1;   // Communications with AOP OK
   MCC3_6A_CommsOK : BOOL := 1;   // Communications with AOP OK
   MCC3_6D_CommsOK : BOOL := 1;   // Communications with AOP OK
   MCC3_6G_CommsOK : BOOL := 1;   // Communications with AOP OK
   MCC3_6J_CommsOK : BOOL := 1;   // Communications with AOP OK
   MCC3_7A_CommsOK : BOOL := 1;   // Communications with AOP OK
   MCC3_7C_CommsOK : BOOL := 1;   // Communications with AOP OK
   MCC3_7E_CommsOK : BOOL := 1;   // Communications with AOP OK
   MCC3_7G_CommsOK : BOOL := 1;   // Communications with AOP OK
   MCC3_7K_CommsOK : BOOL := 1;   // Communications with AOP OK
   MCC3_8A_CommsOK : BOOL;   // Communications with AOP OK
   MCC3_8D_CommsOK : BOOL := 1;   // Communications with AOP OK
   MCC3_8H_CommsOK : BOOL;   // Communications with AOP OK
   MCC3_8K_CommsOK : BOOL := 1;   // Communications with AOP OK
   MCC3_9A_CommsOK : BOOL := 1;   // Communications with AOP OK
   MCC3_9C_CommsOK : BOOL := 1;   // Communications with AOP OK
   MCC3_9E_CommsOK : BOOL := 1;   // Communications with AOP OK
   MCC3_9G_CommsOK : BOOL := 1;   // Communications with AOP OK
   MCC3_9J_CommsOK : BOOL := 1;   // Communications with AOP OK
   MCC3_9L_CommsOK : BOOL;   // Communications with AOP OK
   MCC4_1E_CommsOK : BOOL := 1;   // Communications with AOP OK
   MCC4_2A_CommsOK : BOOL := 1;   // Communications with AOP OK
   MCC4_2C_CommsOK : BOOL := 1;   // Communications with AOP OK
   MCC4_2E_CommsOK : BOOL := 1;   // Communications with AOP OK
   MCC4_2G_CommsOK : BOOL;   // Communications with AOP OK
   MCC4_2K_CommsOK : BOOL := 1;   // Communications with AOP OK
   MCC4_3A_CommsOK : BOOL := 1;   // Communications with AOP OK
   MCC4_3C_CommsOK : BOOL := 1;   // Communications with AOP OK
   MCC4_3E_CommsOK : BOOL := 1;   // Communications with AOP OK
   MCC4_3G_CommsOK : BOOL := 1;   // Communications with AOP OK
   MCC4_3J_CommsOK : BOOL := 1;   // Communications with AOP OK
   MCC4_3L_CommsOK : BOOL := 1;   // Communications with AOP OK
   MCC4_4A_CommsOK : BOOL;   // Communications with AOP OK
   MCC4_4C_CommsOK : BOOL := 1;   // Communications with AOP OK
   MCC4_4E_CommsOK : BOOL;   // Communications with AOP OK
   MCC4_4G_CommsOK : BOOL;   // Communications with AOP OK
   MCC4_4J_CommsOK : BOOL;   // Communications with AOP OK
   MCC4_4L_CommsOK : BOOL;   // Communications with AOP OK
   MCC4_5A_CommsOK : BOOL;   // Communications with AOP OK
   MCC4_5C_CommsOK : BOOL := 1;   // Communications with AOP OK
   MCC4_5E_CommsOK : BOOL;   // Communications with AOP OK
   MCC4_5G_CommsOK : BOOL;   // Communications with AOP OK
   MCC4_5J_CommsOK : BOOL;   // Communications with AOP OK
   MCC4_5L_CommsOK : BOOL;   // Communications with AOP OK
   MotorsControlTag : MotorsControlUDT := (MCC2_2A.Speed := 80, MCC2_2A.Spare := 7892, MCC2_2D.Speed := 80, MCC2_2G.Speed := 80, MCC2_2K.Speed := 80, MCC2_9H.Speed := 56, MCC2_21G.Speed := 80, MCC3_2A.Speed := 80, MCC3_2D.Speed := 80, MCC3_2G.Speed := 80, MCC3_2K.Speed := 80, MCC3_3A.Speed := 80, MCC3_3D.Speed := 80, MCC3_3G.Speed := 80, MCC3_3K.Speed := 80, MCC3_4A.Speed := 80, MCC3_4D.Speed := 30, MCC3_4G.Speed := 80, MCC3_4K.Speed := 80, MCC3_5A.Speed := 80, MCC3_5D.Speed := 80, MCC3_5G.Speed := 80, MCC3_5K.Speed := 80, MCC3_6A.Speed := 33, MCC3_6D.Speed := 32, MCC3_7G.Speed := 50, MCC3_7K.Speed := 56, MCC3_8D.Speed := 57, MCC3_8K.Speed := 55, MCC3_22E.Spare := 3214, MCC4_1E.Speed := 60, MCC4_2G.Speed := 95, MCC4_2K.Speed := 66);   // Only Instance of UDT
   MotorsStatusTag : MotorsStatusUDT := (MCC2_2A.Spare := 12345, MCC2_3C.OverloadPercent := 1, MCC2_3G.OverloadPercent := 3, MCC2_3J.OverloadPercent := 2, MCC2_6A.StatusBits := 4, MCC2_6A.OverloadPercent := 4, MCC2_6A.MSG_FaultWarning := 3, MCC2_7K.StatusBits := 4, MCC2_7K.MSG_FaultWarning := 8, MCC2_8B.StatusBits := 4, MCC2_8B.MSG_FaultWarning := 8, MCC2_8K.StatusBits := 4, MCC2_8K.MSG_FaultWarning := 8, MCC2_10C.StatusBits := 4, MCC2_10C.MSG_FaultWarning := 6, MCC2_11L.StatusBits := 4, MCC2_11L.MSG_FaultWarning := 8, MCC2_13E.StatusBits := 4, MCC2_13E.MSG_FaultWarning := 8, MCC2_14J.StatusBits := 4, MCC2_14J.MSG_FaultWarning := 8, MCC2_20G.StatusBits := 4, MCC2_20G.OverloadPercent := 16, MCC2_20G.MSG_FaultWarning := 8, MCC2_21K.StatusBits := 4, MCC2_21K.MSG_FaultWarning := 8, MCC3_8A.StatusBits := 4, MCC3_8A.MSG_FaultWarning := 8, MCC3_8H.StatusBits := 4, MCC3_8H.MSG_FaultWarning := 8, MCC3_9G.StatusBits := 1, MCC3_9L.StatusBits := 4, MCC3_9L.MSG_FaultWarning := 8, MCC3_10D.StatusBits := 4, MCC3_10D.MSG_FaultWarning := 8, MCC3_10J.StatusBits := 4, MCC3_10J.MSG_FaultWarning := 8, MCC3_11J.StatusBits := 4, MCC3_11J.MSG_FaultWarning := 8, MCC3_12A.StatusBits := 4, MCC3_12A.MSG_FaultWarning := 8, MCC3_14L.StatusBits := 4, MCC3_14L.MSG_FaultWarning := 8, MCC3_15J.StatusBits := 4, MCC3_15J.MSG_FaultWarning := 8, MCC3_16E.StatusBits := 4, MCC3_16E.MSG_FaultWarning := 8, MCC3_18G.StatusBits := 4, MCC3_18G.MSG_FaultWarning := 8, MCC3_22E.Spare := 54321, MCC4_1E.StatusBits := 4, MCC4_1E.MSG_FaultWarning := 9, MCC4_2G.StatusBits := 4, MCC4_2G.MSG_FaultWarning := 8, MCC4_4A.StatusBits := 4, MCC4_4A.MSG_FaultWarning := 8); {access Read Only}   // Only Instance of UDT
   MSG_ReadSpacing_T : TIMER := (PRE := 100, ACC := 92, EN := 1, TT := 1); {access Read Only}   // Read MCC2 & MCC3 Motor Commands From PLC1 Spacing Timer
   OKToRunMotors : BOOL := 1; {access Read Only}   // Messages from PLC1 Ok, OK to run
   ReadMotorError_CTR : COUNTER := (PRE := 4); {access Read Only}   // Read Message form PLC1 Error Counter
   ReadMotorsFromPLC1 : MESSAGE; {access Read Only}   // Read from PLC1, MotorsToPLC2
        MessageParameters(ServiceCode := 16#004c, LocalElement := MotorsControlTag, ...)
   ReadMotorsFromPLC1_DOS : BOOL := 1; {access Read Only}   // Read Motors from PLC1 Done One Shot
END_VAR
